FUNCTION_BLOCK "GCS7_E_DEVC"	// FB 38
TITLE = DevCtrl
//  
//COPYRIGHT:    (C) 2004 BY  BUHLER AG, CH-9240 UZWIL  SWITZERLAND
//
//PRODUCT:      GCS7
//
//TITLE:        Element DevCTRL (Profibus)
//              (GCPROVB Revision 10)
//
//-------------------------------------------------------------------------
//
//IDENT:        AUTHOR:             DEPT:                      DATE:
//FB38.2.1      A.Egli              CT3                        01-Dec-2005
//              Parameter Upload Change DBD86-->DBD88
//FB38.2.0      A.Egli              CT3                        05-Jan-2005
//              Parameter Upload (uses DB10)
//FB38.1.1      A. Egli             CT3                        20-Sep-2004
//              Integration test
//FB38.1.0      A. Egli             CT3                        08-Jun-2004
//              1st Release in S7
//
//-------------------------------------------------------------------------
//
//PURPOSE:      MANUAL : see [DEVCENMAN]
//
//RESTRICTIONS: S7
//
//              (*2) : Not used for MZDE
//
//=======================================================
//Log Message: 
//------------------------------------------------------
//0     = Fault Cannceled
//1..79 = AlarmLC : Alarmnumber see manual of MEAF
//90    = Fault Remote Control
//91    = StStopped
//92    = StDosing
//93    = StEmptied
//94    = Timeout starting
//95    = Wrong value
//96    = Communication fault
//97    = 
//98    = 
//99    = Collected alarm
//
//=======================================================
//StCode:  State               
//------------------------------------------------------
//32    StFault                 
// 1    StStopped                   Stopped
//41    Stopped.HWStop              StStopped + InHWStop 
//51    Stopped.DPFault             StStopped + DPFault
// 2    StStarting              
// 3    StStarted               
// 7    StStopping              
//
//
AUTHOR : EA
FAMILY : GCS7LL
NAME : DEVCTRL
VERSION : 2.1
VAR
  StCode : INT ;	//Element state code
  InEnable : BOOL ;	//Enable to run the element (manual and automatic mode)
  InAutomaticControl : BOOL ;	//1=Automatic Control, 0=Manual Control
  CmdRestart : BOOL ;	//Pulse to send "Newstart" to LC
  InHoldStartValue : BOOL ;	//Is sent to LC : de: Startwert aktiv
  spare0203 : BOOL ;
  spare0205 : BOOL ;
  spare0206 : BOOL ;
  spare0207 : BOOL ;
  CmdOff : BOOL ;	//Pulse to stop the element (manual mode)
  CmdOn : BOOL ;	//Pulse to start the element (manual mode)
  CmdNext : BOOL ;	//Pulse to start the element in automatic mode
  CmdFaultReset : BOOL ;	//Command to reset fault
  InLocal : BOOL ;	//1= Local mode (no fault by start with service switch)
  InManual : BOOL ;	//1= Manual / 0= Automatic
  InReport : BOOL ;	//Report of all state transitions
  spare0307 : BOOL ;
  InHWStop : BOOL ;	//HW stop is detected, no fault
  InDPFault : BOOL ;	//DP-Fault is detected, no fault
  InSimulation : BOOL ;	//MZAH: Simulation with DPSim
  OutComFault : BOOL ;	//Communication fault
  OutWrongValue : BOOL ;	//Wrong nominal values, rejected by MEAF
  OutSteamValueOn : BOOL ;	//de: Dampfventil angesteuert
  OutLS1Closed : BOOL ;	//de: Endschalter 1 geschlossen
  OutLS2Closed : BOOL ;	//de: Endschalter 2 geschlossen
  StStopped : BOOL ;	//Element is stopped
  StStarting : BOOL ;	//Element is starting
  StStarted : BOOL ;	//Element is dosing
  StStopping : BOOL ;	//Element is stopping
  StFault : BOOL ;	//Element has a communication or device fault
  InTemperature : INT ;	//Is sent to LC: Target value [0.1°C]  sent to MEAF
  InSteamValueManual : INT ;	//Is sent to LC: Target value steam control manual mode [0.1%]
  InProductFlowrate : DINT ;	//Is sent to LC: Actual flowrate product [kg/h]
  InStartValueSteam : INT ;	//Is sent to LC: CTRL.START Start value for steam control [0.1%]
  InQMin : INT ;	//Is sent to LC: Minimum dosing value TCON.QMIN
  InQMax : INT ;	//Is sent to LC: Maximum dosing value TCON.QMAX
  spare20 : INT ;
  spare22 : INT ;
  spare24 : INT ;
  spare26 : INT ;
  OutTemperature1 : INT ;	//Is read from LC: [0.1°C]
  OutTemperature2 : INT ;	//Is read from LC: [0.1°C]
  OutTemperature3 : INT ;	//Is read from LC: [0.1°C]
  OutSteamAc : DINT ;	//Is read from LC: Actual flowrate steam [0.1%]
  OutStartValueSteam : DINT ;	//Is read from LC: Start value for steam control [0.1%]
  spare42 : DINT ;	//Is read from LC: Minimum dosing value TCON.QMIN
  spare46 : DINT ;	//Is read from LC: Maximum dosing value TCON.QMAX
  OutAlarmNr : INT ;	//Is read from MEAF
  OutAlarmNrLog : INT ;	//Last textnumber send to log
  InFilter : ARRAY  [0 .. 95 ] OF //These alarms are not printed  (1=no alarm)
  BOOL ;
  Par : STRUCT
   ParObjectNo : INT ;	//Is used for communication with PC, e.g. for message
   ParMsgType : INT ;	//Is used for message (translation of state)
   ParHornCode : INT ;	//Is used by horn module
   ParLogOff : BOOL ;	//Report is off
   ParManual : BOOL ;	//Manual mode wihout interlocking
   ParIOByteNr : INT ;	//PROFIBUS: Address of first input and output byte
   ParMonTime : INT ;	//Monitoring time starting and stopping
   OutMonTime : INT ;	//Monitoring time starting and stopping
   OutHelpFlags : STRUCT 	//Is sent to FBAL
    OutAlarmTimeOut : BOOL ;
    CmdFaultReset : BOOL ;
    OutFaultResetDone : BOOL ;
    OutTestNewAlarm : BOOL ;	//Aux. signal to retry fault message
    OutFlagFaultResetDone : BOOL ;
    OutComFaultRead : BOOL ;
    OutComFaultSend : BOOL ;
    OutRelevantFault : BOOL ;
    OutNoAlarm : BOOL ;	//Alarmnumber 0 is read form LC
   END_STRUCT ;
   Command : STRUCT
    Start : BOOL ;	//de: Start
    Automatic : BOOL ;	//de: Automat/Manual
    Restart : BOOL ;	//de: Neustart mit Startwert und Startzeit
    StartValueActive : BOOL ;	//de: Startwert aktiv
    spare04 : BOOL ;
    spare05 : BOOL ;
    spare06 : BOOL ;
    AcceptNewDataReady : BOOL ;	//FBAL: de: Quittierung neue Werte Bereit
    spare10 : BYTE ;
    spare20 : BYTE ;
    CommandReady : BOOL ;	//de: Steuersignale gültig
    spare31 : BOOL ;
    spare32 : BOOL ;
    spare33 : BOOL ;
    spare34 : BOOL ;
    ResetAlarm : BOOL ;	//de: Alarm löschen
    NewSendData : BOOL ;	//de: Aenderung Sendedaten
    AcceptNewRcvData : BOOL ;	//de: Quittierung Aenderung Empfangsdatensatz
   END_STRUCT ;
   Status : STRUCT
    Operation : BOOL ;	//de: Betrieb
    spare01 : BOOL ;
    RestartDone : BOOL ;	//de: Neustart wurde vorgenommen
    spare03 : BOOL ;
    spare04 : BOOL ;
    spare05 : BOOL ;	//
    spare06 : BOOL ;
    NewDataReady : BOOL ;	//de: Neue Werte Bereit
    SteamValueOn : BOOL ;	//de: Dampfventil angesteuert
    LS1Closed : BOOL ;	//de: Endschalter 1 geschlossen
    LS2Closed : BOOL ;	//de: Endschalter 2 geschlossen
    spare20 : BYTE ;
    spare30 : BOOL ;
    spare31 : BOOL ;
    spare32 : BOOL ;
    RemoteControl : BOOL ;	//de: Sollwertvorgabe Remote
    WrongValue : BOOL ;	//de: Falscher Sollwert
    SumFault : BOOL ;	//de: Sammelalarm
    AcceptNewSendData : BOOL ;	//de: Quittierung Aenderung Sendedaten
    NewRcvData : BOOL ;	//de: Aenderung Empfangsdaten
   END_STRUCT ;
  END_STRUCT ;
END_VAR
VAR_TEMP
  tmpLOGvalue : WORD ;	//LOG value
  tmpCommand : INT ;
  tmpFault : BOOL ;
  tmpOff : BOOL ;
  tmpOn : BOOL ;
  tmpLocal : BOOL ;
  tmpLocalFault : BOOL ;
  tmpReport : BOOL ;
  tmpFlag : BOOL ;
  tmpLenDyn : DINT ;
  tmpAddrOffset : DINT ;
  tmpAddr : WORD ;
  tmpReturn : INT ;
  DPData : STRUCT
   StatusCommand : DWORD ;
   NrSndDataSet : BYTE ;	//de: Nummer Sendedatensatz
   IdxSndDataSet : BYTE ;	//de: Index Sendedatensatz
   NrRcvDataSet : BYTE ;	//de: Nummer Empfangsdatensatz
   IdxRcvDataSet : BYTE ;	//de: Index Empfangsdatensatz
   Data : ARRAY  [1 .. 4 ] OF DINT ;
  END_STRUCT ;
  Set001 : STRUCT
   Temperature1 : INT ;	//Is read from LC: [0.1°C]
   Temperature2 : INT ;	//Is read from LC: [0.1°C]
   Temperature3 : INT ;	//Is read from LC: [0.1°C]
   StreamAc : DINT ;	//Is read from LC: Actual flowrate steam [0.1%]
   StartValueSteam : INT ;	//Is read from LC: Start value for steam control [0.1%]
   DosingValueMax : INT ;	//Is read from LC: Maximum dosing value TCON.QMAX
   DosingValueMin : BYTE ;	//Is read from LC: Minimum dosing value TCON.QMIN
   AlarmNr : BYTE ;	//Is read from MEAF
  END_STRUCT ;
  Set128 : STRUCT
   Temperature : INT ;	//Is sent to LC: Target value [0.1°C]  sent to MEAF
   SteamValueManual : INT ;	//Is sent to LC: Target value steam control manual mode [0.1%]
   spare12 : INT ;	//Is sent to LC: Target value steam control manual mode [0.1%]
   FlowrateProdAc : DINT ;	//Is sent to LC: Actual flowrate product [kg/h]
   StartValueSteam : INT ;	//Is sent to LC: CTRL.START Start value for steam control [0.1%]
   DosingValueMax : INT ;	//Is sent to LC: Maximum dosing value TCON.QMAX
   DosingValueMin : INT ;	//Is sent to LC: Minimum dosing value TCON.QMIN
  END_STRUCT ;
END_VAR
BEGIN
NETWORK
TITLE =  Start Global
      L     90;
      T     #tmpLenDyn;	//--> Len dynamic data in byte
      TAR2;
      L     DW#16#FFFFFF;
      AD;
      T     #tmpAddrOffset;
NETWORK
TITLE = PC Control
//=== Test Object number =====================
      L     "SYS_DirectCtrlDB".PC.ObjectNo;	//PCControl.ObjectNo
      L     #Par.ParObjectNo;	//Input ObjectNo
      <>I;
      JC    Ctrl;
//=== Test OType      ========================
      L     1138;	//Input object type
      L     "SYS_DirectCtrlDB".PC.ObjectType;	//PCControl.ObjectType
      <>I;
      JC    Ctrl;
//=== Test Handshake =========================
      A     "SYS_DirectCtrlDB".PC.Hsk.FExamine;	//Handshake.FExamine
      JC    pExa;
      A     "SYS_DirectCtrlDB".PC.Hsk.FDefineCmd;	//Handshake.FDefineCmd
      JC    pCmd;
      A     "SYS_DirectCtrlDB".PC.Hsk.FDefinePara;	//Handshake.FDefinePara
      JC    pPar;
pIni: L     2;	//FcInit
      UC    "SYS_DirectCtrl";
      JU    Ctrl;
//Write parameter 
pPar: NOP   0;
//Write new commands from PC to Interface of group 
pCmd: A     "SYS_DirectCtrlDB".PC.Cmd1[2];	//Cmd1[2]  =CmdRestart
      S     #CmdRestart;
      A     "SYS_DirectCtrlDB".PC.Cmd1[8];	//Cmd1[8]  =CmdOff
      S     #CmdOff;
      A     "SYS_DirectCtrlDB".PC.Cmd1[9];	//Cmd1[9]  =CmdOn
      S     #CmdOn;
      A     "SYS_DirectCtrlDB".PC.Cmd1[10];	//Cmd1[10] =CmdNext
      S     #CmdNext;
      A     "SYS_DirectCtrlDB".PC.Cmd1[11];	//Cmd1[11] =CmdFaultReset
      S     #CmdFaultReset;
      A     "SYS_DirectCtrlDB".PC.Cmd1[13];	//Cmd1[13] =CmdManualOn
      S     #InManual;
      A     "SYS_DirectCtrlDB".PC.Cmd2[13];	//Cmd2[13] =CmdManualOff
      R     #InManual;
      A     "SYS_DirectCtrlDB".PC.Cmd1[14];	//Cmd1[14] =CmdReportOn
      S     #InReport;
      A     "SYS_DirectCtrlDB".PC.Cmd2[14];	//Cmd2[14] =CmdReportOff
      R     #InReport;
//Define Value
      AN    "SYS_DirectCtrlDB".PC.Hsk.FDefineValue;	// PC.Hsk.FDefineValue
      ON    #InManual;
      JC    pIni;
      JU    pIni;
pExa: TAR2;	//Address dynamic datas
      T     "SYS_DirectCtrlDB".GC.InDynAddr;	//-->PCControl.GC.InDynAddr
      L     #tmpLenDyn;	//Length dynamic datas
      T     "SYS_DirectCtrlDB".GC.InDynLen;	//-->PCControl.GC.InDynLen
      L     0;
      T     "SYS_DirectCtrlDB".GC.InParaAddr;	//-->PCControl.GC.InParaAddr
      T     "SYS_DirectCtrlDB".GC.InParaLen;	//-->PCControl.GC.InParaLen
      L     1;	//Code FcExamine
      UC    "SYS_DirectCtrl";
      L     10;	//Revision
      T     "SYS_DirectCtrlDB".GC.Revision;
Ctrl: NOP   0;
NETWORK
TITLE = (Profibus) Read data and store Data 
      L     #Par.ParIOByteNr;
      T     #tmpAddr;
      A     #InSimulation;
      JC    rSim;
      CALL  "SIEMENS_DPRD_DAT" (
           LADDR                    := #tmpAddr,
           RET_VAL                  := #tmpReturn,
           RECORD                   := #DPData);
      L     #tmpReturn;
      L     0;
      <>I;
      =     #Par.OutHelpFlags.OutComFaultRead;
      JC    rcv0;
      JU    rDP;
//read from Simulation
rSim: R     #Par.OutHelpFlags.OutComFaultRead;
      A     "GCS7_Gr_SimDPtoImage";
      L     P#I 0.0;
      JC    rDB1;
      OPN   "TEST_IOSimuliInput";
      L     P#DBX 0.0;
rDB1: L     #Par.ParIOByteNr;
      SLD   3;
      +D;
      LAR1;
      L     D [AR1,P#0.0];
      T     #DPData.StatusCommand;
      L     B [AR1,P#4.0];
      T     #DPData.NrSndDataSet;
      L     B [AR1,P#5.0];
      T     #DPData.IdxSndDataSet;
      L     B [AR1,P#6.0];
      T     #DPData.NrRcvDataSet;
      L     B [AR1,P#7.0];
      T     #DPData.IdxRcvDataSet;
      L     D [AR1,P#8.0];
      T     #DPData.Data[1];
      L     D [AR1,P#12.0];
      T     #DPData.Data[2];
      L     D [AR1,P#16.0];
      T     #DPData.Data[3];
      L     D [AR1,P#20.0];
      T     #DPData.Data[4];
//==Copy Status===============
rDP:  L     #DPData.NrRcvDataSet;
      L     0;
      ==I;
      JC    R001;
      CALL  "SIEMENS_BLKMOV" (
           SRCBLK                   := #DPData.StatusCommand,
           RET_VAL                  := #tmpReturn,
           DSTBLK                   := #Par.Status);
      AN    #Par.Status.NewRcvData;
      A     #InSimulation;
      JC    rcv0;
//===============================
//Answer Dataset 001
      L     #DPData.NrRcvDataSet;
      L     1;
      <>I;
      JC    r11;	//[2.0]
      CALL  "SIEMENS_BLKMOV" (
           SRCBLK                   := #DPData.Data,
           RET_VAL                  := #tmpReturn,
           DSTBLK                   := #Set001);
      L     #Set001.Temperature1;
      T     #OutTemperature1;
      L     #Set001.Temperature2;
      T     #OutTemperature2;
      L     #Set001.Temperature3;
      T     #OutTemperature3;
      L     #Set001.StreamAc;
      T     #OutSteamAc;
      L     #Set001.StartValueSteam;
      T     #OutStartValueSteam;
//Reset old alarm flags with CmdFaultReset
      A     #Par.OutHelpFlags.OutFlagFaultResetDone;
      A     "SYS_Pulse1000ms";
      R     #Par.OutHelpFlags.OutFlagFaultResetDone;
      R     #Par.OutHelpFlags.OutFaultResetDone;
      S     #Par.OutHelpFlags.OutTestNewAlarm;
      L     0;
      L     #Set001.AlarmNr;
      ==I;
      =     #Par.OutHelpFlags.OutNoAlarm;
//  keep old alalrm number
      A     #Par.OutHelpFlags.OutNoAlarm;
      A     #Par.OutHelpFlags.OutRelevantFault;
      AN    #Par.OutHelpFlags.OutTestNewAlarm;
      AN    #InLocal;
      AN    #InManual;
      JC    rA1;
      T     #OutAlarmNr;
rA1:  JU    R11;	//[2.0]   
//===============================
//[2.0]--> LC Parameter 
//Reading dataset 11
R11:  L     "SYS_DirectCtrlLCDB".PC.ObjectNo;
      L     #Par.ParObjectNo;
      <>I;
      JC    R127;
      AN    "SYS_DirectCtrlLCDB".PC.Hsk.FExamineFirst;
      AN    "SYS_DirectCtrlLCDB".PC.Hsk.FExamineNext;
      JC    R127;
// -- Start Reading with Dataset 11
      L     11;
      T     #DPData.NrRcvDataSet;
      L     253;	//First
      A     "SYS_DirectCtrlLCDB".PC.Hsk.FExamineFirst;
      JC    rLC9;
      L     254;	//Next
rLC9: T     #DPData.IdxRcvDataSet;
      JU    rcv0;
//---Answer  dataset 11 ---
//---Answer  dataset 12 ---
r11:  L     #DPData.NrRcvDataSet;
      L     11;
      <>I;
      JC    rLCB;
// Answer Dataset 11
      L     '  ';
      T     "SYS_DirectCtrlLCDB".PC.Value[1];
      L     #DPData.Data[1];
      T     DB10.DBD 60;
      L     #DPData.Data[2];
      T     DB10.DBD 64;
      L     #DPData.Data[3];
      T     DB10.DBD 68;
      L     #DPData.Data[4];
      T     DB10.DBD 72;
      L     #DPData.IdxRcvDataSet;
      L     255;
      ==I;
      JC    rLCE;
      S     "SYS_DirectCtrlLCDB".GC.Set11Done;
      L     12;
      T     #DPData.NrRcvDataSet;
      L     0;
      T     #DPData.IdxRcvDataSet;
      JU    rcv0;	//--> Read dataset 12
// Answer Dataset 12
rLCB: L     #DPData.NrRcvDataSet;
      L     12;
      <>I;
      JC    r127;
      L     #DPData.Data[1];
      T     DB10.DBD 76;
      L     #DPData.Data[2];
      T     DB10.DBD 80;
      L     #DPData.Data[3];
      T     DB10.DBD 84;
      L     #DPData.Data[4];
      T     DB10.DBD 88;
      AN    "SYS_DirectCtrlLCDB".GC.Set11Done;
      JC    R127;
rLCE: L     12;
      CALL  "SYS_DirectCtrl";
      JU    R127;
//<--[2.0]
//===============================
//Answer  dataset 127
r127: L     #DPData.NrRcvDataSet;
      L     127;
      <>I;
      JC    r001;
      JU    R001;
//===============================
//Else Read Dataset 1
r001: JU    R001;	// =no valide answer read dataset 001
//===============================
//Read Dataset 001
R001: L     1;
      T     #DPData.NrRcvDataSet;
      L     0;
      T     #DPData.IdxRcvDataSet;
      A     #Par.OutHelpFlags.OutFaultResetDone;
      AN    "SYS_Pulse1000ms";
      S     #Par.OutHelpFlags.OutFlagFaultResetDone;
      JU    rcv0;
//===============================
//Read Dataset 127
R127: L     127;
      T     #DPData.NrRcvDataSet;
      L     0;
      T     #DPData.IdxRcvDataSet;
      JU    rcv0;
//===============================
rcv0: NOP   0;
NETWORK
TITLE = (Profibus) Status to ASW
      A     #Par.OutHelpFlags.OutComFaultRead;
      O     #Par.OutHelpFlags.OutComFaultSend;
      =     #OutComFault;
      A     #Par.Status.SteamValueOn;
      AN    #OutComFault;
      =     #OutSteamValueOn;
      A     #Par.Status.LS1Closed;
      AN    #OutComFault;
      =     #OutLS1Closed;
      A     #Par.Status.LS2Closed;
      AN    #OutComFault;
      =     #OutLS2Closed;
//=======================================
//Init in local mode  
//=======================================
      AN    #InLocal;
      AN    #InManual;
      ON    #OutComFault;
      JC    alJL;
      L     0;
      T     #OutSteamAc;
alJL: NOP   0;
NETWORK
TITLE =  All State Init
//===Clear tmp Variable
//===Global Group Orders===
      A     "GCS7_Gr_OutManualOn";	//Global.OutManualOn
      S     #InManual;
      A     "GCS7_Gr_OutManualOff";	//Global.OutManualOff
      R     #InManual;
      A     #InManual;
      S     "GCS7_Gr_InManual";	//Global.InManualMode
//---Report is on---
      O     "GCS7_Gr_OutReportAll";	//---Global OutReportAll
      O     #InReport;
      =     #tmpReport;
//---FaultReset is on---
      A     "GCS7_Gr_OutFaultReset";	//Gr.OutFaultReset
      S     #CmdFaultReset;
//---State---
//---Local---
      A     #InLocal;
      AN    #InManual;
      =     #tmpLocalFault;
      A     #tmpLocalFault;
      O     #InHWStop;
      O     #InDPFault;
      =     #tmpLocal;
//---Off---
      AN    #InManual;
      ON    #Par.ParManual;
      AN    #InEnable;
      O     #tmpLocal;
      O     #CmdOff;
      =     #tmpOff;
//---On---
      A     #CmdNext;
      AN    #InManual;
      O     #CmdOn;
      AN    #tmpOff;
      =     #tmpOn;
//--- Time out---
      AN    #StStarting;
      AN    #StStopping;
      AN    #StFault;
      R     #Par.OutHelpFlags.OutAlarmTimeOut;
      JC    inJ1;
      A     #Par.OutHelpFlags.OutAlarmTimeOut;
      O     #StFault;
      JC    inJ1;
      L     0;
      L     #Par.OutMonTime;
      >I;
      =     #Par.OutHelpFlags.OutAlarmTimeOut;
      AN    "GCS7_Gr_OutTick200ms";	// Global Tick 200ms
      JC    inJ1;
      +     -2;	// Decrement all 200ms
      T     #Par.OutMonTime;
inJ1: NOP   0;
//=======================================
//Fault   
//=======================================
      A     #Par.Status.WrongValue;
      =     #OutWrongValue;
//--- Fault   
      LAR1  #tmpAddrOffset;
      L     P##InFilter;
      +AR1;	//Pointer to #InFilter
      L     #OutAlarmNr;
      +AR1;	//Pointer to #InFilter[OutAlarmNumber]
      L     #OutAlarmNr;
      L     0;
      <>I;
      AN    DIX [AR1,P#0.0];	//#InFilter[OutAlarmNumber]
      O;
      A     #Par.Status.SumFault;
      AN    #InFilter[0];
      =     #Par.OutHelpFlags.OutRelevantFault;
      A     #Par.OutHelpFlags.OutRelevantFault;
      A     #Par.Status.SumFault;
      O     #OutComFault;
      O     #Par.OutHelpFlags.OutAlarmTimeOut;
      O     #Par.Status.WrongValue;
      ON    #Par.Status.RemoteControl;
      AN    #tmpLocal;
      =     #tmpFault;
NETWORK
TITLE = (Profibus) Prepare Command for MEAF
      A     #Par.Command.Start;
      =     #tmpFlag;
      A     #tmpOn;
      S     #Par.Command.Start;
      A     #StFault;
      O     #tmpOff;
      O     #StStopping;
      R     #Par.Command.Start;
//==============================
      A     #InAutomaticControl;
      =     #Par.Command.Automatic;
//================================
      A     #CmdRestart;
      S     #Par.Command.Restart;
      A     #CmdRestart;
      A     #Par.Command.Restart;
      A     #Par.Status.RestartDone;
      R     #Par.Command.Restart;
      R     #CmdRestart;
//================================
      A     #InHoldStartValue;
      =     #Par.Command.StartValueActive;
//==============================
      A     #Par.Status.AcceptNewSendData;
      A     #Par.Command.ResetAlarm;
      R     #Par.Command.ResetAlarm;
      S     #Par.OutHelpFlags.OutFaultResetDone;
      A     #CmdFaultReset;
      AN    #Par.Status.AcceptNewSendData;
      R     #CmdFaultReset;
      S     #Par.Command.ResetAlarm;
      R     #Par.OutHelpFlags.OutAlarmTimeOut;
//==============================
      A     #Par.Status.NewDataReady;
      =     #Par.Command.AcceptNewDataReady;
//==============================
      SET;
      =     #Par.Command.CommandReady;
//==============================
      A     #Par.Status.NewRcvData;
      =     #Par.Command.AcceptNewRcvData;
//==============================
      AN    #Par.Status.AcceptNewSendData;
      =     #Par.Command.NewSendData;
NETWORK
TITLE = (Profibus) Send Data
//======================================================
//Test Send Dataset 000 done
      L     #DPData.NrSndDataSet;
      L     0;
      <>I;
      JC    s128;
      JU    S128;	//-->send 128
//------------------------------------------------
//Test Send Dataset 128 done
s128: L     #DPData.NrSndDataSet;
      L     128;
      <>I;
      JC    S000;	//-->Send 000
      JU    S128;	//-->Send 128
//==================================================
//Send Dataset 128
S128: L     128;
      T     #DPData.NrSndDataSet;
      L     0;
      T     #DPData.IdxSndDataSet;
      L     #InTemperature;
      T     #Set128.Temperature;
      L     #InSteamValueManual;
      T     #Set128.SteamValueManual;
      L     0;
      T     #Set128.spare12;
      L     #InProductFlowrate;
      T     #Set128.FlowrateProdAc;
      L     #InStartValueSteam;
      T     #Set128.StartValueSteam;
      L     #InQMax;
      T     #Set128.DosingValueMax;
      L     #InQMin;
      T     #Set128.DosingValueMin;
      JU    send;
//======================================================
//Send Dataset 0
S000: L     0;
      T     #DPData.NrSndDataSet;
      L     0;
      T     #DPData.IdxSndDataSet;
send: CALL  "SIEMENS_BLKMOV" (
           SRCBLK                   := #Par.Command,
           RET_VAL                  := #tmpReturn,
           DSTBLK                   := #DPData.StatusCommand);
      CALL  "SIEMENS_BLKMOV" (
           SRCBLK                   := #Set128,
           RET_VAL                  := #tmpReturn,
           DSTBLK                   := #DPData.Data);
      A     #InSimulation;
      JC    sSim;
      CALL  "SIEMENS_DPWR_DAT" (
           LADDR                    := #tmpAddr,
           RECORD                   := #DPData,
           RET_VAL                  := #tmpReturn);
      L     #tmpReturn;
      L     0;
      <>I;
      =     #Par.OutHelpFlags.OutComFaultSend;
      JU    DP_C;
//write to Simulation
sSim: R     #Par.OutHelpFlags.OutComFaultSend;
      A     "GCS7_Gr_SimDPtoImage";
      L     P#Q 0.0;
      JC    rDB2;
      OPN   "TEST_IOSimuliOutput";
      L     P#DBX 0.0;
rDB2: L     #Par.ParIOByteNr;
      SLD   3;
      +D;
      LAR1;
      L     #DPData.StatusCommand;
      T     D [AR1,P#0.0];
      L     #DPData.NrSndDataSet;
      T     B [AR1,P#4.0];
      L     #DPData.IdxSndDataSet;
      T     B [AR1,P#5.0];
      L     #DPData.NrRcvDataSet;
      T     B [AR1,P#6.0];
      L     #DPData.IdxRcvDataSet;
      T     B [AR1,P#7.0];
      L     #DPData.Data[1];
      T     D [AR1,P#8.0];
      L     #DPData.Data[2];
      T     D [AR1,P#12.0];
      L     #DPData.Data[3];
      T     D [AR1,P#16.0];
      L     #DPData.Data[4];
      T     D [AR1,P#20.0];
DP_C: NOP   0;
NETWORK
TITLE = States
//===State machine===
      A     #StStopped;
      JC    S0;
      A     #StStarting;
      JC    S1;
      A     #StStarted;
      JC    S2;
      A     #StStopping;
      JC    S3;
      A     #StFault;
      JC    S4;
      S     #StStopped;	//Init
      JU    S0;
NETWORK
TITLE =  StStopped
xxS0: S     #StStopped;
      R     #StStarted;
      JU    LOGX;
S0:   A     #tmpFault;
      R     #StStopped;
      JC    xxS4;	//--> Transition to StFault
      A     #Par.Status.Operation;
      AN    #OutComFault;
      O     #Par.Command.Start;
      R     #StStopped;
      JC    xxS1;	//--> Transition to StStarting
      JU    OUT;
NETWORK
TITLE =  StStarting
xxS1: S     #StStarting;
      R     #Par.OutHelpFlags.OutAlarmTimeOut;
      L     #Par.ParMonTime;
      T     #Par.OutMonTime;
      JU    OUT;
S1:   A     #tmpFault;	//Condition for StFault
      R     #StStarting;
      JC    xxS4;	//--> Transition to StFault
      A     #tmpOff;
      R     #StStarting;
      JC    xxS3;	//--> Transition to StStopping
      A     #Par.Status.Operation;
      R     #StStarting;
      JC    xxS2;	//--> Transition to StStarted
      JU    OUT;
NETWORK
TITLE =  StStarted
xxS2: S     #StStarted;
      JU    LOGX;
S2:   A     #tmpFault;	//Condition for StFault/StFalse
      R     #StStarted;
      JC    xxS4;	//--> Transition to StFault
      A     #tmpOff;
      ON    #Par.Status.Operation;
      R     #StStarted;
      JC    xxS3;	//--> Transition to StStopping
      JU    OUT;
NETWORK
TITLE =  StStopping
xxS3: S     #StStopping;
      R     #Par.OutHelpFlags.OutAlarmTimeOut;
      L     #Par.ParMonTime;
      T     #Par.OutMonTime;
      A     #StFault;
      R     #StFault;
      JC    LOGC;	//-->Message Operator ('fault cancelled' )
//State StStopping
S3:   A     #tmpFault;
      AN    #tmpLocal;
      R     #StStopping;
      JC    xxS4;	//-->Transition to StFault
      A     #tmpOn;
      R     #StStopping;
      JC    xxS1;	//-->Transition to StStarting 
      AN    #Par.Status.Operation;
      O     #OutComFault;
      R     #StStopping;
      JC    xxS0;	//-->Transition to StStopped 
      JU    OUT;
NETWORK
TITLE =  FAULT
// State Fault
S4:   AN    #tmpFault;	//---Condition for StStopping
      A     #Par.OutHelpFlags.OutTestNewAlarm;
      O     #tmpLocalFault;
      JC    xxS3;	// Transition to StStopping
      A     #Par.OutHelpFlags.OutTestNewAlarm;
      JC    xxS4;
      JU    OUT;
NETWORK
TITLE = LOG
xxS4: S     "GCS7_Gr_InFaultFlag";	//Gr.InFaultFlag
      S     #StFault;
      R     #Par.OutHelpFlags.OutFaultResetDone;
      R     #Par.OutHelpFlags.OutTestNewAlarm;
      CALL  "SYS_Horn_Code" (
           FcCode                   := 1,
           ParObjectType            := 1138,
           ParObjectNo              := #Par.ParObjectNo,
           ParHornCode              := #Par.ParHornCode);
      L     #Par.ParMonTime;
      T     #Par.OutMonTime;
//Alarm Communication
      L     B#(1, 96);
      A     #OutComFault;
      JC    LOG;
//Tiemout
      A     #Par.OutHelpFlags.OutAlarmTimeOut;
      L     B#(1, 94);	// Message ('fault timeout')
      JC    LOG;
//Alarm-Nr 1..80
      L     0;
      L     #OutAlarmNr;
      ==I;
      JC    LOG2;
      L     B#(1, 0);
      OW;
      JU    LOG;	//Alarms 1..80
//Fault Remote Control
LOG2: L     B#(1, 90);	// Message ('fault DP Mode')   //[5.2]
      AN    #Par.Status.RemoteControl;	//[5.2]
      JC    LOG;	//[5.2]
//Fault Wrong Value
      A     #Par.Status.WrongValue;
      L     B#(1, 95);	// Message ('fault wrong value')
      JC    LOG;
//Collected Alarm
      L     B#(1, 99);	// Message ('fault collected alarm')
      JU    LOG;
//===============================================
//State Transition
LOGX: AN    #tmpReport;
      JC    OUT;
      A     #StStopped;
      L     B#(4, 91);	//Message ('Stopped')
      JC    LOG;
      A     #StStarted;
      L     B#(4, 92);	//Message ('Started')
      JC    LOG;
      JU    OUT;
LOGC: L     B#(4, 0);	//Message ('fault cancelled')
LOG:  A     #Par.ParLogOff;	//---Set LOG Message
      JC    OUT;
      T     #tmpLOGvalue;
      L     W#16#FF;
      AW;
      T     #OutAlarmNrLog;
      CALL  "GCS7_LogConvert" (
           ObjectNo                 := #Par.ParObjectNo,
           MsgType                  := #Par.ParMsgType,
           ClassMsgTxt              := #tmpLOGvalue,
           OType                    := 1138);	//LOG Message Converter / Entry / Contains Class and TextNo
NETWORK
TITLE = Global End
OUT:  SET;	//---Clear all commands
      R     #CmdOff;
      R     #CmdOn;
      R     #CmdNext;
//--Output for group 
      AN    #InLocal;
      O     #InManual;
      A     #InDPFault;
      S     "GCS7_Gr_InDPFault";
      AN    #InLocal;
      O     #InManual;
      A     #InHWStop;
      S     "GCS7_Gr_InHWStop";
NETWORK
TITLE = State Code
//--Stopped, Substate ---
      AN    #StStopped;
      JC    STC2;
      L     41;	//Code: StStopped.HWStop
      A     #InHWStop;
      JC    STC;
      L     51;	//Code: StStopped.DPFault
      A     #InDPFault;
      JC    STC;
      L     1;	// Code: stopped
      JC    STC;
//--------------------
STC2: L     2;	//Code: StStarting
      A     #StStarting;
      JC    STC;
      L     3;	//Code: StStarted
      A     #StStarted;
      JC    STC;
      L     7;	//Code: StStopping
      A     #StStopping;
      JC    STC;
      L     32;	//Code: fault
STC:  L     #StCode;	//Old state code
      TAK;
      T     #StCode;	//Save state code
      <>I;
      L     3;	//Load code for CBit methode
      CC    "SYS_CBitCtrl";
END_FUNCTION_BLOCK

FUNCTION_BLOCK "GCS7_E_MYFA_MOZD"	// FB 39
TITLE = MYFA-MOZD
//  
//COPYRIGHT:    (C) 1997  BUHLER AG, CH-9240 UZWIL, SWITZERLAND
//
//PRODUCT:      GCS7
//
//TITLE:        Element Control MYFA-MOZD or MOZD (Liquid Regulator)
//
//-------------------------------------------------------------------------
//
//IDENT:        AUTHOR:             DEPT:                       DATE:
//
//FB39.3.0      A. Egli             CT3                         17-Jun-2002
//              New Release with one block
//              MOZD or MYFA-MOZD  
//FB39.2.1      A. Egli             CT3                         11-Oct-1999
//              M12.2 "Gr.OutCmdNext removed
//FB39.2A       A. Egli             CT3                         04-Mai-1998
//              StFault = StCode 32
//FB39.1A       A.Egli              AEE61                       25-Jul-1997
//              1st Release in S7
//
//-------------------------------------------------------------------------
//
//PURPOSE:      MANUAL : see [MYFxxMAN]
//
//RESTRICTIONS: S7
//              ACCU2: Pointer to dynamic datas of the element
//              ACCU1: Pointer to parameter datas of the element
//
//-------------------------------------------------------------------------
//=======================================================
//Log Message: 
//------------------------------------------------------
// 0   stopped
// 1   started
// 9   fault cancelled
//10   fault MYFA
//11   fault analog input
//12   fault set value
//
//=======================================================
//StCode:  State               
//------------------------------------------------------
//32   StFault                 
// 1   StStopped               
//41   StStopped.HWStop           StStopped + InHWStop 
//51   StStopped.DPFault          StStopped + DPFault
// 3   StStarted               
//
AUTHOR : EA
FAMILY : GCS7LL
NAME : MYFAMOZD
VERSION : 3.0
VAR
  StCode : INT ;	//Element state code
  InEnable : BOOL ;	//Enable to run
  spare0201 : BOOL ;
  spare0202 : BOOL ;
  spare0203 : BOOL ;
  spare0204 : BOOL ;
  CmdNewJob : BOOL ;	//Pulse to erase OutWtTotalWater
  InRemote : BOOL ;	//Target flowrate for MOZD from PLC
  InpLcOk : BOOL ;	//Digital input 1=MOZD ok / 0=MOZD Alarm
  CmdOff : BOOL ;	//Pulse to start in manual mode
  CmdOn : BOOL ;	//Pulse to stop in manual mode
  CmdNext : BOOL ;	//Start next element (Automatic mode)
  CmdFaultReset : BOOL ;	//Command to reset fault
  InLocal : BOOL ;	//1= Local mode
  InManual : BOOL ;	//1= Manual/ 0= Automatic
  InReport : BOOL ;	//Report of all state transitions
  spare0307 : BOOL ;
  InHWStop : BOOL ;	//HW stop is detected, no fault
  InDPFault : BOOL ;	//DP-Fault is detected, no fault
  OutFaultAI : BOOL ;	//Fault analog input
  OutFaultSetValue : BOOL ;	//Set value out of range
  spare0404 : BOOL ;
  spare0405 : BOOL ;
  OutpRemote : BOOL ;	//Digital output flowrate water from PLC
  spare0407 : BOOL ;
  StStopped : BOOL ;	//Element is stopped
  spare0501 : BOOL ;
  StStarted : BOOL ;	//Element is started
  spare0503 : BOOL ;
  StFault : BOOL ;	//Element has a fault
  InpFlowrateWater : INT ;	//Analog input actual flowrate water [digits]
  MYFA : STRUCT 	//With MYFA
   InMoisture : INT ;	//Moisture target value [0.1 %]
   InpFlowrateProduct : INT ;	//Analog input actual flowrate product [digits]
   InpMoisture : INT ;	//Analog input actual moisture [digits]
   OutMoisture : INT ;	//Moisture actual value [0.1 %]
   OutFlowrateProduct : INT ;	//Flowrate product actual value in [kg/h]
   OutpMoisture : INT ;	//Analog output to target moisture [digits]
  END_STRUCT ;
  MOZD : STRUCT 	//Without MYFA
   InOutFlowrateWaterPpm : INT ;	//Flowrate water target value [0.0 to 10.0%]
   InOutFlowrateWater : INT ;	//Flowrate water target value [dl/h]
   InFlowrateProduct : INT ;	//Flowrate product actual value in [kg/h]
   OutpFlowrateWater : INT ;	//Analog output target flowrate water
   OutpFlowrateProduct : INT ;	//Analog output flowrate product
  END_STRUCT ;
  OutFlowrateWater : INT ;	//Flowrate water actual value in [dl/h]
  OutTotalWater : DINT ;	//Total feeded weight water   [dl]
  OutAlarmNrLog : INT ;	//Last textnumber send to log
  Par : STRUCT
   ParObjectNo : INT ;	//Is used for communication with PC, e.g. for message
   ParMsgType : INT ;	//Is used for message (translation of state)
   ParHornCode : INT ;	//Is used by horn module
   ParLogOff : BOOL ;	//Report is off
   ParManual : BOOL ;	//Manual mode without interlocking
   ParWago : BOOL ;	//Wago analog module format
   ParMYFA : BOOL ;
   ParInFlowrateWaterPc : BOOL ;	//Target value flowrate water from group in Pc
   ParOutFlowrateWaterPc : BOOL ;	//Analog output flowrate water in [0.0 to 10.0%]
   ParFlowrateWater100Pc : INT  := 20000;	//Flowrate water   by 100 % of analog value [dl/h]
   ParFlowrateProduct100Pc : INT  := 30000;	//Flowrate product by 100 % of analog value [kg/h]
   OutCorrectionWeight : REAL ;	//Correction weight for calcuation of OutWtTotalWater [kg]
   spare16 : DINT ;
  END_STRUCT ;
END_VAR
VAR_TEMP
  tmpLOGvalue : WORD ;	//LOG value
  tmpReport : BOOL ;	//Global LOG all
  tmpEnable : BOOL ;
  tmpLenDyn : DINT ;
  tmpEndTime : BOOL ;
  tmpLocal : BOOL ;
  tmpFault : BOOL ;
  tmpFlowWater : REAL ;
  tmpMaxDigits : REAL ;	//ParWago=0: 27'648 / ParWago=1: 32'767
  tmpLocalFault : BOOL ;
END_VAR
BEGIN
NETWORK
TITLE =  Start Global
      L     58;
      T     #tmpLenDyn;	//--> Len dynamic data in byte
NETWORK
TITLE = PC Control
//=== Test Object number =====================
      L     "SYS_DirectCtrlDB".PC.ObjectNo;	//PCControl.ObjectNo
      L     #Par.ParObjectNo;	//Input ObjectNo
      <>I;
      JC    Ctrl;
//=== Test OType      ========================
      L     1039;	//Input object type
      L     "SYS_DirectCtrlDB".PC.ObjectType;	//PCControl.ObjectType
      <>I;
      JC    Ctrl;
//=== Test Handshake =========================
      A     "SYS_DirectCtrlDB".PC.Hsk.FExamine;	// Handshake.FExamine
      JC    pExa;
      A     "SYS_DirectCtrlDB".PC.Hsk.FDefineCmd;	// Handshake.FDefineCmd
      JC    pCmd;
      A     "SYS_DirectCtrlDB".PC.Hsk.FDefinePara;	// Handshake.FDefinePara
      JC    pPar;
pIni: L     2;	// FcInit
      UC    "SYS_DirectCtrl";
      JU    Ctrl;
// Write parameter 
pPar: NOP   0;
// Write new commands from PC to Interface of group 
pCmd: A     "SYS_DirectCtrlDB".PC.Cmd1[8];	//Cmd1[8] =CmdOff
      S     #CmdOff;
      A     "SYS_DirectCtrlDB".PC.Cmd1[9];	//Cmd1[9] =CmdOn
      S     #CmdOn;
      A     "SYS_DirectCtrlDB".PC.Cmd1[10];	//Cmd1[10] =CmdNext
      S     #CmdNext;
      A     "SYS_DirectCtrlDB".PC.Cmd1[11];	//Cmd1[11] =CmdFaultReset
      S     #CmdFaultReset;
      A     "SYS_DirectCtrlDB".PC.Cmd1[13];	//Cmd1[13] =CmdManualOn
      S     #InManual;
      A     "SYS_DirectCtrlDB".PC.Cmd2[13];	//Cmd2[13] =CmdManualOff
      R     #InManual;
      A     "SYS_DirectCtrlDB".PC.Cmd1[14];	//Cmd1[14] =CmdReportOn
      S     #InReport;
      A     "SYS_DirectCtrlDB".PC.Cmd2[14];	//Cmd2[14] =CmdReportOff
      R     #InReport;
      JU    pIni;
pExa: TAR2;	// Address Dynamic datas
      T     "SYS_DirectCtrlDB".GC.InDynAddr;	// -->PCControl.GC.InDynAddr
      L     #tmpLenDyn;	// Length Dynamic datas
      T     "SYS_DirectCtrlDB".GC.InDynLen;	// -->PCControl.GC.InDynLen
      L     0;
      T     "SYS_DirectCtrlDB".GC.InParaAddr;	// -->PCControl.GC.InParaAddr
      T     "SYS_DirectCtrlDB".GC.InParaLen;	// -->PCControl.GC.InParaLen
      L     1;	// Code FcExamine
      UC    "SYS_DirectCtrl";
      L     10;	//Revision
      T     "SYS_DirectCtrlDB".GC.Revision;
NETWORK
TITLE =  All State Init
//===Clear tmp Variable
//===Global Group Orders===
Ctrl: A     "GCS7_Gr_OutManualOn";	//Gr.OutManualOn
      S     #InManual;
      A     "GCS7_Gr_OutManualOff";	//Gr.OutManualOff
      R     #InManual;
      A     #InManual;
      S     "GCS7_Gr_InManual";	//Gr.InManual
//---Local---
      A     #InLocal;
      AN    #InManual;
      =     #tmpLocalFault;
      A     #tmpLocalFault;
      O     #InHWStop;
      O     #InDPFault;
      =     #tmpLocal;
//---Report is on---
      A     "GCS7_Gr_OutReportAll";	//Gr.OutReportAll
      O     #InReport;
      =     #tmpReport;
//---tmpEnable---
      A     #InEnable;
      AN    #InLocal;
      AN    #InManual;
      O(;
      A     #InEnable;
      O     #Par.ParManual;
      A     #InManual;
      );
      AN    #CmdOff;
      =     #tmpEnable;
//---tmpFault---
      L     #MOZD.InOutFlowrateWater;
      L     #Par.ParFlowrateWater100Pc;
      >D;
      O(;
      L     #MOZD.InFlowrateProduct;
      L     #Par.ParFlowrateProduct100Pc;
      >D;
      );
      AN    #Par.ParMYFA;
      O(;
      L     #MYFA.InMoisture;
      L     200;
      >I;
      A     #Par.ParMYFA;
      );
      =     #OutFaultSetValue;
      A     #OutFaultAI;	//Overflow analog input
      ON    #InpLcOk;
      O     #OutFaultSetValue;
      =     #tmpFault;
      A     #InRemote;
      =     #OutpRemote;
//---tmpMaxDigits
      L     2.764800e+04;	//Siemens fullrange MaxDigits
      AN    #Par.ParWago;
      JC    Ctr2;
      L     3.276700e+04;	//Wago fullrange MaxDigits
Ctr2: T     #tmpMaxDigits;
NETWORK
TITLE = States
//===State machine===
      A     #StStopped;
      JC    S0;
      A     #StStarted;
      JC    S2;
      A     #StFault;
      JC    S4;
      S     #StStopped;	// Init
      JU    S0;
NETWORK
TITLE = StStopped
// Any transition to StClosed
xxS0: S     #StStopped;
      AN    #InReport;
      JC    OUT;
      L     B#(4, 0);	// Message ('stopped' )
      JU    LOG;
//=== Logic ====
//Transition to StStarted 
S0:   A     #CmdNext;
      AN    #InManual;
      A     #tmpEnable;
      O;
      A     #CmdOn;
      A     #InManual;
      A     #tmpEnable;
      R     #StStopped;
      JC    xxS2;
//Transition to StFault 
      A     #tmpFault;
      AN    #tmpLocal;
      R     #StStopped;
      JC    xxS4;
      JU    OUT;
NETWORK
TITLE = StStarted
// Any transition to StStarted
xxS2: S     #StStarted;
      S     #StStarted;
      AN    #tmpReport;
      JC    OUT;
      L     B#(4, 1);	// Message ('started')
      JU    LOG;
//=== Logic ====
//Transition to StStopped
S2:   AN    #tmpEnable;
      R     #StStarted;
      JC    xxS0;
// Transition to StFault
      A     #tmpFault;
      AN    #tmpLocal;
      R     #StStarted;
      JC    xxS4;
      JU    OUT;
NETWORK
TITLE = StFault
// Any transiton to Fault  
xxS4: S     "GCS7_Gr_InFaultFlag";	// Gr.InFaultFlag
      S     #StFault;
      CALL  "SYS_Horn_Code" (
           FcCode                   := 1,
           ParObjectType            := 1039,
           ParObjectNo              := #Par.ParObjectNo,
           ParHornCode              := #Par.ParHornCode);
      A     #OutFaultAI;	//Overflow analog input
      L     B#(1, 11);	// Message ('fault analag input' )
      JC    LOG;
      A     #OutFaultSetValue;
      L     B#(1, 12);	//Message ('fault set value' )
      JC    LOG;
      L     B#(1, 10);	// Message ('fault MYFA' )
      JU    LOG;
//=== Logic ====
S4:   AN    #CmdFaultReset;
      AN    "GCS7_Gr_OutFaultReset";	//Gr.OutFaultReset
      AN    #tmpLocal;
      JC    OUT;
// retry of fault message
      A     #tmpFault;
      AN    #tmpLocal;
      JC    xxS4;
      R     #StFault;
      S     #StStopped;
      L     B#(3, 9);	// Message ('fault cancelled' )
      JU    LOG;
NETWORK
TITLE = Log
LOG:  A     #Par.ParLogOff;	//---Set LOG Message
      JC    OUT;
      T     #tmpLOGvalue;
      L     W#16#FF;
      AW;
      T     #OutAlarmNrLog;
      CALL  "GCS7_LogConvert" (
           ObjectNo                 := #Par.ParObjectNo,
           MsgType                  := #Par.ParMsgType,
           ClassMsgTxt              := #tmpLOGvalue,
           OType                    := 1039);	// LOG Message Converter / Entry / Contains Class and TextNo
OUT:  NOP   0;
      SET;
      R     #OutFaultAI;	//--> Overflow analog input
NETWORK
TITLE = MOZD: Calculate target flowrate Water 
      A     #Par.ParInFlowrateWaterPc;
      JC    fwPc;
      L     #MOZD.InOutFlowrateWater;	//[dl/h]
      DTR;
      L     #MOZD.InFlowrateProduct;	//[kg/h]
      DTR;
      /R;
      L     1.000000e+02;	//0.1 *1000                  
      *R;
      RND;
      T     #MOZD.InOutFlowrateWaterPpm;	//-->Target flowrate water in [0.1%] 
      JU    fwJ0;
fwPc: L     #MOZD.InFlowrateProduct;
      DTR;
      L     #MOZD.InOutFlowrateWaterPpm;
      DTR;
      *R;
      L     1.000000e+02;
      /R;
      RND;
      T     #MOZD.InOutFlowrateWater;	//--> Target flowrate water
NETWORK
TITLE = MOZD: Calculate Analog Output value flow water
fwJ0: L     0;
      AN    #StStarted;
      ON    #OutpRemote;
      JC    fwJ1;
      AN    #Par.ParOutFlowrateWaterPc;
      JC    fwJ2;
// Analog output: Unit = 0..10%
      L     #MOZD.InOutFlowrateWaterPpm;	// dl/h
      DTR;	// Integer to real
      L     1.000000e+02;	// 10.0% 
      <=R;
      JC    fwJ3;
      L     1.000000e+00;	// 100%          
      JU    fwJ4;
// Analog output: Unit = dl/h
fwJ2: L     #MOZD.InOutFlowrateWater;	// dl/h
      DTR;	// Integer to real
      L     #Par.ParFlowrateWater100Pc;
      DTR;	// Integer to real
      <=R;
      JC    fwJ3;
      L     1.000000e+00;	// 100%          
      JU    fwJ4;
fwJ3: /R;
fwJ4: L     #tmpMaxDigits;	// Units maximum         
      *R;
      RND;	// Real to Integer
fwJ1: T     #MOZD.OutpFlowrateWater;
NETWORK
TITLE = MOZD:Calculate Analog Output flowrate product
      L     0;
      AN    #StStarted;
      JC    fpJ1;
      L     #MOZD.InFlowrateProduct;	//  kg/h
      DTR;	// Integer to real
      L     #Par.ParFlowrateProduct100Pc;
      DTR;	// Integer to real
      <=R;
      JC    fpJ2;
      L     1.000000e+00;	// 100%          
      JU    fpJ3;
fpJ2: /R;
fpJ3: L     #tmpMaxDigits;	// Units maximum         
      *R;
      RND;	// Real to Integer
fpJ1: T     #MOZD.OutpFlowrateProduct;
NETWORK
TITLE = Calculate actual flowrate water
      L     -32767;
      L     #InpFlowrateWater;	//  kg/h
      >=I;
      AN    #Par.ParWago;	// Fault only with Siemens analog input
      S     #OutFaultAI;	//--> Overflow analog input
      L     0.000000e+00;
      JC    ai0;
      L     #InpFlowrateWater;	//  kg/h
      DTR;	// Integer to real
      L     #tmpMaxDigits;	// Units maximum         
      /R;
      L     #Par.ParFlowrateWater100Pc;
      DTR;	// Integer to real
      *R;
ai0:  T     #tmpFlowWater;
      RND;	// Real to Integer
      T     #OutFlowrateWater;
NETWORK
TITLE = Calculate Analog Output moisture
      L     0;
      AN    #StStarted;
      ON    #OutpRemote;
      JC    msJ1;
      L     #MYFA.InMoisture;	//[0.1%]
      DTR;	// Integer to real
      L     2.000000e+02;
      <=R;
      JC    msJ3;
      L     1.000000e+00;	// 100%          
      JU    msJ4;
msJ3: /R;
msJ4: L     #tmpMaxDigits;	// Units maximum         
      *R;
      RND;	// Real to Integer
msJ1: T     #MYFA.OutpMoisture;
NETWORK
TITLE = Calculate actual moisture
      L     -32767;
      L     #MYFA.InpMoisture;	//  
      >=I;
      AN    #Par.ParWago;	// Fault only with Siemens analog input
      S     #OutFaultAI;	//--> Overflow analog input
      L     0.000000e+00;
      JC    aim0;
      L     #MYFA.InpMoisture;	//  
      DTR;	// Integer to real
      L     #tmpMaxDigits;	// Units maximum         
      /R;
      L     2.000000e+02;
      *R;
aim0: RND;	// Real to Integer
      T     #MYFA.OutMoisture;
NETWORK
TITLE = BOTH: Calculate actual flowrate product
      L     -32767;
      L     #MYFA.InpFlowrateProduct;
      >=I;
      AN    #Par.ParWago;	// Fault only with Siemens analog input
      S     #OutFaultAI;	//--> Overflow analog input
      L     0.000000e+00;
      JC    aip0;
      L     #MYFA.InpFlowrateProduct;
      DTR;	// Integer to real
      L     #tmpMaxDigits;	// Units maximum         
      /R;
      L     #Par.ParFlowrateProduct100Pc;
      DTR;	// Integer to real
      *R;
aip0: RND;	// Real to Integer
      T     #MYFA.OutFlowrateProduct;
NETWORK
TITLE = BOTH: Calculate OutWtTotal
      AN    #CmdNewJob;
      JC    wtJ1;
      L     0;
      T     #OutTotalWater;
      L     0.000000e+00;
      T     #Par.OutCorrectionWeight;
      JU    clJ1;
wtJ1: AN    "GCS7_Gr_OutTick1s";	//Gr.OutTick1s
      JC    clJ1;
      L     #tmpFlowWater;
      L     3.600000e+03;	// [3600s]  
      /R;
      L     #Par.OutCorrectionWeight;
      +R;
      T     #Par.OutCorrectionWeight;
      RND-;
      L     #OutTotalWater;
      +D;
      T     #OutTotalWater;
      L     #Par.OutCorrectionWeight;
      L     #Par.OutCorrectionWeight;
      RND-;
      DTR;	// Integer to Real
      -R;
      T     #Par.OutCorrectionWeight;	//New rest 
NETWORK
TITLE = Global End
//---Clear all commands
clJ1: SET;
      R     #CmdOn;
      R     #CmdOff;
      R     #CmdNewJob;
      R     #CmdNext;
      R     #CmdFaultReset;
//--Output for group 
      A     #InDPFault;
      AN    #tmpLocalFault;
      S     "GCS7_Gr_InDPFault";
      A     #InHWStop;
      AN    #tmpLocalFault;
      S     "GCS7_Gr_InHWStop";
      A     #StFault;
      S     "GCS7_Gr_InFault";	// Gr.InFault
NETWORK
TITLE = State Code
//--Stopped, Substate ---
      AN    #StStopped;
      JC    STC2;
      L     41;	//Code: StStopped.HWStop
      A     #InHWStop;
      JC    STC;
      L     51;	//Code: StStopped.DPFault
      A     #InDPFault;
      JC    STC;
      L     1;	//Code: stopped
      A     #StStopped;
      JC    STC;
//===============
STC2: L     3;	// Code: started
      A     #StStarted;
      JC    STC;
      L     32;	// Code: fault
STC:  L     #StCode;	// Old state code
      TAK;
      T     #StCode;	// Save state code
      <>I;
      L     3;	// Load code for CBit methode
      CC    "SYS_CBitCtrl";
END_FUNCTION_BLOCK

FUNCTION_BLOCK "GCS7_E_Scale"	// FB 40
TITLE = Scale DIFF/DUMP
//  
//COPYRIGHT:    (C) 1996  BUHLER AG, CH-9240 UZWIL, SWITZERLAND
//
//PRODUCT:      GCS7
//
//TITLE:        Element Control Scale DIFF, DUMP, with OPTO22 or DP
//
//-------------------------------------------------------------------------
//
//IDENT:        AUTHOR:             DEPT:                       DATE:
//FB40.7.8      A. Egli             BASE                        29-Jan-2009
//              - DUMP Check InPreCutoffWeight and Status.TotalReached       
//FB40.7.7      Ph. Engler          GP92                        16-Jun-2008
//              - No failure with MEAG-Fault 17       
//              - Transition from StEmptying to StStarting when
//                InOutRestDischargeBin has been reset
//FB40.7.6      A. Egli             BASE                        09-Apr-2008
//              Disable Alarm 18 Battery Low
//FB40.7.5      A. Egli             CT3                         25-Mai-2007
//              - Overflow weight OutNotErasableWeight is 999'999'999 
//FB40.7.4      A.Egli              CT3                         20-Feb-2006
//              For CmdRefill test also tmpOn: Tested by P.Engler
//FB40.7.3      A.Egli              CT3                         01-Dec-2005
//              Parameter Upload Change DBD86-->DBD88
//FB40.7.2      A.Egli              CT3                         17-Mai-2005
//              Reset Flowrate only when OutComFault=1 
//FB40.7.1      A.Egli              CT3                         14-Mar-2005
//              Read Status.TotalReached only with data set 1
//FB40.7.0      A.Egli              CT3                         05-Jan-2005
//              Parameter Upload (uses DB10)
//FB40.6.6      Ph. Engler          MU664                       13-Sep-2004
//              -DIFF: Command.Restdischarge only in LCStep=1
//FB40.6.5      A.Egli              CT3                         23-Jul-2004
//              DUMP: Transition StDosing to StSopped also in LCStep=2
//FB40.6.4      A.Egli              CT3                         18-Mai-2004
//              DUMP: Transition to Started, when Level uncovered
//FB40.6.3      A.Egli              CT3                         24-Mar-2004
//              Replace T D [AR1,xxx] with T LD [AR1,xxx]
//FB40.6.2      A.Egli              CT3                         17-Nov-2003
//              - Alarm 90: Fault Remote Control
//              - MEAF: Ignor SumFault
//              - Local Mode: ComFault change to StStopped
//              - Manual mode: Set EnableEmptying
//FB40.6.1      A. Egli             CT3                         19-Mai-2003
//              Use Status.Operation as condtion for stopped
//FB40.6.0      A. Egli             CT3                         17-Jun-2002
//              New Release with one block
//              OPTO22 and Profibus   
//              LC Alarm 14 (DPFault) =Log Text number 12
//              InRecipeNr=Byte21
//FB40.5.1      P.Engler            CT3                         22-Mai-2002
//              Transition StStopped to StEmptying
//FB40.5.0      K.Tischer           CT3                         20-Sep-2001
//              Several modifications for MEAF
//FB40.4.3      K.Tischer           CT3                         02-Aug-2001
//              InSeqStopDUMP: S/R #OutStateTarget.EmptyingDUMP [4.3]
//FB40.4.2      A.Egli              CT3                         25-Jun-2001
//              par.OutLCAlarm.NoProduct replaced par.OutLCAlarm.NoProduct
//              Reset CmdRefill        
//FB40.4.1      P.Müller            MU664                       16-Mar-2001
//              Wait in StStarting until LCStep <> 1 removed
//FB40.4.0      S. Kalberer         CT3                         28-Nov-2000
//              Emptying event and signals adapted (MEAF V32B)
//FB40.3.0      A. Egli             CT3                         14-Jul-2000
//              New command MEAF
//FB40.2.6      A. Egli             CT3                         17-Mar-2000
//              Length for answer telegram
//FB40.2.4      S. Kalberer         CT3                         18-Feb-2000
//              CmdNewJob: Clear scale total in StDosing by OutStopPoint
//FB40.2.3      S. Kalberer         CT3                         11-Feb-2000
//              Relog fault, store OutState.InDischarged
//              CmdNewJob: immediate clear OutWtJobActual
//FB40.2C       S. Kalberer         CT3                         24-Sep-1999
//              Powerfailure dependency eliminated
//              ParManual behaviour corrected
//FB40.2B       S. Kalberer         CT3                         10-Mar-1999
//              MEAF compatible interface
//FB40.2A       A. Egli             CT3                         04-Mai-1998
//              StFault = StCode 32
//FB40.1A       A.Egli              AEE61                       28-Jul-1997
//              1st Release in S7
//
//-------------------------------------------------------------------------
//
//PURPOSE:      MANUAL : see [SCALExxMAN]
//
//RESTRICTIONS: S7
//              ACCU2: Pointer to dynamic datas of the element
//              ACCU1: Pointer to parameter datas of the element
//
//=======================================================
//Log Message: 
//------------------------------------------------------
//0     = Fault Cannceled
//1..79 = AlarmLC : Alarmnumber see manual of MEAF
//90    = Fault Remote Control
//91    = StStopped
//92    = StDosing
//93    = StEmptied
//94    = Timeout starting
//95    = WrongValue
//96    = Communication fault
//97    = 
//98    = 
//99    = Collected alarm
//
//=======================================================
//StCode:  State               
//------------------------------------------------------
//32   StFault                 
// 1   StStopped               
//41   StStopped.HWStop              StStopped + InHWStop 
//51   StStopped.DPFault             StStopped + DPFault
// 2   StStarting              
// 3   StDosing                
// 9   StEmptying              
//10   StEmptied               
//11   StRefill                
AUTHOR : EA
FAMILY : GCS7LL
NAME : SCALE
VERSION : 7.8
VAR
  StCode : INT ;	//Element state code
  InEnable : BOOL ;	//Enable to run scale
  InOutRestdischargeScale : BOOL ;	//Fully emptying scale (MEAF-DIFF)
  InDisableDischargeDUMP : BOOL ;	//stop discharge DUMP Scale
  InRestDosing : BOOL ;	//Restdosing (only MEAF)
  CmdNewValue : BOOL ;	//Send new taregt value to scale
  CmdNewJob : BOOL ;	//Clear actual weight or restart in state StEmptied
  CmdRefill : BOOL ;	//Refill of scale after maintenance (MEAF-DIFF)
  InOutRestdischargeBin : BOOL ;	//Fully emptying bin and scale (MEAF-DIFF + DUMP)
  CmdOff : BOOL ;	//Pulse to stop scale (manual mode)
  CmdOn : BOOL ;	//Pulse to start scale(manual mode)
  CmdNext : BOOL ;	//Start next element  (automatic mode)
  CmdFaultReset : BOOL ;	//Command to reset fault
  InLocal : BOOL ;	//1= Local mode (no fault by start with service switch)
  InManual : BOOL ;	//1= Manual/ 0= Automatic
  InReport : BOOL ;	//Report of all state transitions
  InSeqStopDUMP : BOOL ;	//Sequence stop scale by fully emptying scale (MEAF-DUMP)
  InHWStop : BOOL ;	//HW stop is detected, no fault
  InDPFault : BOOL ;	//DP-Fault is detected, no fault
  InSimulation : BOOL ;	//Simulation with DPSim
  OutComFault : BOOL ;	//Communication fault
  OutDepotEmpty : BOOL ;	//Alarm "DepotEmpty" is set (MEAF-DIFF)
  OutRefillDone : BOOL ;	//Refill is done (MEAF-DIFF)
  OutEmptied : BOOL ;	//Emptying is done
  OutpEnable : BOOL ;	//Output signale for scale
  StStopped : BOOL ;	//Element is stopped
  StStarting : BOOL ;	//Element is starting
  StDosing : BOOL ;	//Element is started, ready for dosing
  StEmptying : BOOL ;	//Emptying is active
  StFault : BOOL ;	//Element has a fault
  StEmptied : BOOL ;	//Element is emptied
  StRefill : BOOL ;	//Refill of the scale (MEAF-DIFF)
  spare57 : BOOL ;
  OutStopPoint : BOOL ;	//Target weight reached
  OutWeightCleared : BOOL ;	//Erasable weight is cleared
  OutWrongValue : BOOL ;	//Wrong nominal values, rejected by MEAF
  InFlowrate : DINT ;	//Is send to LC
  InJobWeight : DINT ;	//Is send to LC
  InRecipeNr : INT ;	//Is send to LC (DIFF only)
  InPreCutoffWeight : INT ;	//Pre cutoff weight
  OutFlowrate : DINT ;	//Is read from LC
  OutJobWeight : DINT ;	//Is calculated by element out of not erasable weight
  OutTotalWeight : DINT ;	//Is read from LC
  OutScaleWeight : DINT ;	//Is read from LC
  OutRecipeNr : INT ;	//Is read from LC (DIFF only)
  OutLCStep : INT ;	//Is read from LC
  OutAlarmNr : INT ;	//Is read from LC
  spare : DINT ;
  OutAlarmNrLog : INT ;	//Last textnumber send to log
  DUMP : STRUCT 	//DUMP only (is only sent, if InDumpWt >0)
   InDumpWeight : INT ;	//de: Schüttgrösse (only Profibus DP)
   InFlowrateLowLimit : INT ;	//de: Untere Leistungsgrenze
   InFlowrateHighLimit : INT ;	//de: Obere Leistungsgrenze
   spare : DINT ;
  END_STRUCT ;
  RecipeDiff : STRUCT 	//Recipe Diff Scale (Profibus only)
   InRecipeNr : INT ;	//Recipe to read or write (DIFF only)
   CmdSend : BOOL ;	//1= Send Dataset 136
   CmdRead : BOOL ;	//1= Read Dataset 136
   OutSendDone : BOOL ;	//Send is done
   OutReadDone : BOOL ;	//Read is done
   OutWrongValue : BOOL ;	//MEAF has recipe rejected
   InOutCutoffWeight : INT ;	//DIFF: Pre cutoff weight
   InOutDensity : INT ;	//DIFF: de: spezifisches Gewicht
   InOutFactor : INT ;	//DIFF: de: Verstaerkungsfaktor Dosiergeschwindigkeit
   InOutAutoCorrFactor : INT ;	//DIFF: de: Automatischer Korrektur Verstaerkungsfaktor
   spare : DINT ;
  END_STRUCT ;
  Par : STRUCT
   ParObjectNo : INT ;	//Is used for communication with PC, e.g. for message
   ParMsgType : INT ;	//Is used for message (translation of state)
   ParHornCode : INT ;	//Is used by horn module
   ParLogOff : BOOL ;	//Report is off
   ParManual : BOOL ;	//Manual mode without interlocking
   ParDUMP : BOOL ;	//1= MEAF:DUMP (MWEE)/ 0=MEAF:DIFF (MWEG,MWEY)
   ParOPTO22 : BOOL ;	//1= OPTO22 / 0= Profibus
   ParNoStep : BOOL ;	//OPTO22: Do not read command 'c' (MWEG1, MWEJ)
   ParMEAF : BOOL ;	//OPTO22: Use new MEAF commands, not compatible to old electronics
   ParFilter : STRUCT 	//Filter to alarm 1=Ignore alarm
    SumFault : BOOL ;	//All: de: Sammelalarm
    A05_24VToLow : BOOL ;	//All:
    A07ADRange : BOOL ;
    A08ADCalibration : BOOL ;
    A09ADFunction : BOOL ;
    A10ADSupply : BOOL ;
    A11AnalogInput : BOOL ;
    AxxCommunication : BOOL ;	//A12: Serial Interface ; A14=DPFault
    A13RemoteControl : BOOL ;
    A16Printer : BOOL ;
    A20NoStandStill : BOOL ;
    A21EmptyingTime : BOOL ;
    A22ScaleOpen : BOOL ;
    A23LLScaleHopper : BOOL ;
    A24WeightHopper : BOOL ;
    A25FrequenceConverter : BOOL ;
    A26Tolerance : BOOL ;
    A27Measurment : BOOL ;
    A28Feeddrive : BOOL ;
    A29FeedingTime : BOOL ;
    A30ZeroTara : BOOL ;
    A32InletSlideGate : BOOL ;
    A33AirPressure : BOOL ;
    A34NoProduct : BOOL ;
   END_STRUCT ;
   ParComDB : INT ;	//OPTO22: Communication DB
   ParLCIdx : INT ;	//OPTO22: Index of data record
   ParLCAddr : INT ;	//OPTO22: Address of LC
   ParIOByteNr : INT ;	//PROFIBUS: Address of first input and output byte Profibus DP
   ParMonTime : INT ;	//After this time the scale must be in the requested state (New)
   Spare90 : DINT ;
   Spare94 : DINT ;
   OutMonTime : INT ;
   OutScaleType : INT ;	//Is read from LC
   OutNotErasableWeight : DINT  := L#-1;	//Is read from LC
   HelpFlags : STRUCT 	//Aux. signal to retry fault message
    CmdNewValue : BOOL ;
    CmdNewJob : BOOL ;
    OutFaultResetDone : BOOL ;
    OutTestNewAlarm : BOOL ;
    CmdSend129 : BOOL ;	//Send of datablock 129 is requested
    OutFlagFaultResetDone : BOOL ;
    OutTargetSnd : BOOL ;
    OutStepRcv : BOOL ;
    OutAlarmTimeOut : BOOL ;
    EnableDosing : BOOL ;	//Help flag for immediate stop
    OutRelevantFault : BOOL ;
    OutNoAlarm : BOOL ;	//Alarmnumber 0 is read form LC
    OutComFaultRead : BOOL ;
    OutComFaultSend : BOOL ;
   END_STRUCT ;
   Command : STRUCT 	//Command for LC, is send to LC
    Start : BOOL ;	//de: Start
    ResetWtTotal : BOOL ;	//de: Total löschen
    RestDischarge : BOOL ;	//de: Restentleeren
    RestDosing_Refill : BOOL ;	//de: DUMP Restdosieren ; DIFF Refill
    EnableEmptying : BOOL ;	//de: Entleerfreigabe
    OverwriteLL : BOOL ;	//de: DIFF: Kein Alarm bei Leerstand
    spare06 : BOOL ;
    AcceptNewDataReady : BOOL ;	//de: Quittierung neue Werte Bereit
    spare10 : BYTE ;
    spare20 : BYTE ;
    CommandReady : BOOL ;	//de: Steuersignale gültig
    spare41 : BOOL ;
    spare42 : BOOL ;
    spare43 : BOOL ;
    spare44 : BOOL ;
    ResetAlarm : BOOL ;	//de: Alarm löschen
    NewSendData : BOOL ;	//de: Aenderung Sendedaten
    AcceptNewRcvData : BOOL ;	//de: Quittierung Aenderung Empfangsdatensatz
   END_STRUCT ;
   Status : STRUCT 	//MEAF DIFF
    Operation : BOOL ;	//de: Betrieb
    TotalReached : BOOL ;	//de: Total erreicht
    RestDischargeDone : BOOL ;	//de: Restentleeren ausgefüht
    PreCutoffWt_ReadyDosing : BOOL ;	//de: DUMP:Vorabschaltpunkt erreicht/DIFF:Dosierbereit
    TotalReady : BOOL ;	//de: Total bereit
    EnableFeeding_Empty : BOOL ;	//de: DUMP:Transportfreigabe/DIFF:Vordepot leer
    WeightPulse : BOOL ;	//de: Gewichtsimpuls
    NewDataReady : BOOL ;	//de: Neue Werte Bereit
    OutOfTolerance_LL : BOOL ;	//de: DUMP: Ausserhalb Leistungstoleranz/DIFF: Leerstand Waage
    _Dosingtime : BOOL ;	//de: DUMP: not used/DIFF: Dosierzeit ueberschritten
    _ZeroTolerance : BOOL ;	//de: DUMP: not used/DIFF: Niveau
    _RefillRequest : BOOL ;	//de: DUMP: not used/DIFF: Produktzufuehrung
    spare14 : BOOL ;
    spare15 : BOOL ;
    spare16 : BOOL ;
    spare17 : BOOL ;
    spare20 : BYTE ;
    Powerfailure : BOOL ;	//DIFF de: Power failure (only with old electronics)
    spare31 : BOOL ;
    spare32 : BOOL ;	//de: Stuerung Remote
    RemoteControlDP : BOOL ;	//de: Sollwertvorgabe Remote
    WrongValue : BOOL ;	//de: Falscher Sollwert
    SumFault : BOOL ;	//de: Sammelalarm
    AcceptNewSendData : BOOL ;	//de: Quittierung Aenderung Sendedaten
    NewRcvData : BOOL ;	//de: Aenderung Empfangsdaten
   END_STRUCT ;
   ComFlags : STRUCT 	//Flags for communication
    c_Done : BOOL ;	//step
    f_Done : BOOL ;	//Alarm, flowrate, actual weight (MEAF:DUMP)
    g_Done : BOOL ;	//Not erasible weight
    r_Done : BOOL ;	//Actual status
    t_Done : BOOL ;	//scale type
    w_Done : BOOL ;	//scale weight    (MEAF:DIFF)
    d_Done : BOOL ;	//Actual value 2  (MEAF:DIFF)
    h_Done : BOOL ;	//only MEAF
    U_Done : BOOL ;	//Lower  flow rate       (MEAF:DUMP)
    O_Done : BOOL ;	//Limit  upper flow rate (MEAF:DUMP)
    M_Done : BOOL ;	//Target weight
    Q_Done : BOOL ;	//Target flow rate
    S_Done : BOOL ;	//Target status 1
    TT_Done : BOOL ;	//Target status 2 (MEAF:DIFF)
    A_Done : BOOL ;	//Commands MEAF
    p_Done : BOOL ;	//not used
    PP_Done : BOOL ;	//not used
    CC_Done : BOOL ;	//C: DumpWt  (MEAF:DUMP)
   END_STRUCT ;
  END_STRUCT ;
END_VAR
VAR_TEMP
  tmpLOGvalue : WORD ;	//LOG value
  tmpCommand : INT ;
  tmpFBNO : INT ;	//Number of the actual FB
  tmpReport : BOOL ;	//Global LOG all
  tmpFault : BOOL ;
  tmpLocal : BOOL ;
  tmpClearCmdFlag : BOOL ;	//Clear pattern Commands
  tmpOn : BOOL ;
  tmpOff : BOOL ;
  tmpSeqStopDUMP : BOOL ;
  tmpWeight : DINT ;
  tmpLenDyn : DINT ;
  tmpAddrOutComFlags : DWORD ;	//Pointer to OutComFlags
  tmpComDB : INT ;
  tmpLocalFault : BOOL ;
  tmpAddrOffset : DINT ;
  tmpImmediateStop : BOOL ;
  tmpFilter : ARRAY  [0 .. 100 ] OF BOOL ;
  tmpAlarmDUMP : STRUCT 	//Is read from DUMP with command f
   Tolerance : BOOL ;	//Tolerance (not on collective alarm)
   SumFault : BOOL ;	//de: Sammelalarm ab V26A
   spare12 : BOOL ;	//n.w.
   ProbeScaleHopper : BOOL ;	//Probe scale hopper   -->alarm 23
   ScaleOpen : BOOL ;	//Scale open -->alarm 22
   StandStill : BOOL ;	//no standstill -->alarm 20
   EmptyingTime : BOOL ;	//emptying time -->alarm 21
   ADConverter : BOOL ;	//AD converter -->alarm 9
  END_STRUCT ;
  tmpAlarmDIFF : STRUCT 	//Is read from DIFF with command d
   DepotEmpty : BOOL ;	//Surge hopper empty (not on collect alarm) --> alarm 34
   ScaleEmpty : BOOL ;	//de: Leerstand Waage (no product)
   Discharger : BOOL ;	//DIFF a2 Frequency converter or feeding drive -->alarm 25
   Tolerance : BOOL ;	//DIFF a2 Tolerance --> alarm 26
   SumFault : BOOL ;	//de: Sammelalarm ab V26A
   TaraPos : BOOL ;	//DIFF a1 n.w.  -->alarm 30
   ADConverter : BOOL ;	//DIFF a1 AD converter--> alarm 9
   Reading : BOOL ;	//DIFF a1 Measuring fault --> alarm 27
  END_STRUCT ;
  tmpCommand_r : STRUCT 	//Is read from DUMP with command r
   Remote : BOOL ;	//MEAF DUMP: r1 Overiding operation
   DischargeDone : BOOL ;	//de: Restentleeren ausgefüht
   WtTotalReached : BOOL ;	//de: Total erreicht
  END_STRUCT ;
  tmpCommand_d : STRUCT 	//Is read from DIFF with command d
   log_1 : BOOL ;	//de: Always 1
   local : BOOL ;	//de: Local Operation
   DischargeDone : BOOL ;	//de: Restentleeren ausgefüht
   Cycle : BOOL ;	//de: Alters the state after every cycle
   Powerfailure : BOOL ;	//de: Power failure
   Operation : BOOL ;	//de: Betrieb (only with old electronic)
   WtTotalReached : BOOL ;	//de: Total erreicht
   ReadyDosing : BOOL ;	//de: Ready for Feeding
  END_STRUCT ;
  tmpCommand_S_DIFF : STRUCT 	//Command are sent to DIFF with command  S
   ResetPowerfailure : BOOL ;	//de:Stromausfallflg löschen
   EnableDosing : BOOL ;	//de: Dosierfreigabe
   ResetWtTotal : BOOL ;	//de: Total löschen
   Bit3 : BOOL ;	//not used
  END_STRUCT ;
  tmpCommand_T : STRUCT 	//Command are sent to DIFF with command  S and T
   Refill : BOOL ;	//fill up
   Emptying : BOOL ;	//discharge
   Bit2 : BOOL ;	//not used
   Bit3 : BOOL ;	//not used
  END_STRUCT ;
  tmpCommand_S_DUMP : STRUCT 	//Command are sent to DUMP with command  S
   RestDosing : BOOL ;	//de: Redsosieren ab V32B
   EnableDosing : BOOL ;	//de: Dosierfreigabe
   ResetWtTotal : BOOL ;	//de: Total löschen
   Emptying : BOOL ;	//de: Restentleeren
  END_STRUCT ;
  tmpCommand_A : STRUCT 	//Is send to MEAF with Command A
   ResetDischarge : BOOL ;	//DIFF:discharge       DUMP:Rest feeding
   StopDischarge_Restdosing : BOOL ;	//DIFF:Stop discharge  DUMP:Rest discharge
   Refill : BOOL ;	//DIFF:Fill up         DUMP:not used
   spare23 : BOOL ;	//
   Start : BOOL ;	//
   Stop : BOOL ;	//
   ResetWtTotal : BOOL ;	//de: Total löschen
   ResetAlarm : BOOL ;
   spare40 : BOOL ;	//
   spare41 : BOOL ;	//
   spare42 : BOOL ;	//
   Modify : BOOL ;	//DIFF/DUMP take over data
   spare30 : BOOL ;	//
   spare31 : BOOL ;	//
   spare32 : BOOL ;	//
   Modify2 : BOOL ;	//
  END_STRUCT ;
  tmpStatus_h_DUMP : STRUCT
   PreCutoffWt : BOOL ;	//de: Vorabschaltgewicht erreicht
   DischargeDone : BOOL ;	//de: Restentleeren ausgefüht
   spare22 : BOOL ;	//not used
   SumFault : BOOL ;	//de: Sammelalarm ab V26A
   Remote : BOOL ;	//de:
   NewDataReady : BOOL ;	//de: Neue Werte Bereit
   WtTotalReached : BOOL ;	//de: Total erreicht
   Tolerance : BOOL ;	//de: Ausserhalb Toleranz
  END_STRUCT ;
  tmpStatus_h_DIFF : STRUCT
   DischargeDone : BOOL ;	//de: Restentleeren ausgefüht
   BufferHopperEmpty : BOOL ;	//de: Vordepot leer
   ReadyDosing : BOOL ;	//de: Dosierbereit
   SumFault : BOOL ;	//de: Sammelalarm ab V26A
   Remote : BOOL ;	//de:
   NewDataReady : BOOL ;	//de: Neue Werte Bereit
   WtTotalReached : BOOL ;	//de: Total erreicht
   ScaleEmpty : BOOL ;	//de: Leerstand Waage (no product)
  END_STRUCT ;
  tmpAddr : WORD ;
  tmpReturn : INT ;
  Set136 : STRUCT
   Density : INT ;	//DIFF: de: spezifisches Gewicht
   Factor : INT ;	//DIFF: de: Verstaerkungsfaktor Dosiergeschwindigkeit
   CutoffWt : INT ;	//Pre cutoff weight
   spare14 : DINT ;
   spare18 : DINT ;
   spare22 : BYTE ;
   AutoCorrFactor : BYTE ;	//DIFF: de: Automatischer Korrektur Verstaerkungsfaktor
  END_STRUCT ;
  Set001 : STRUCT
   FlowrateAc : DINT ;	//de: Istleistung kg/h
   WtTotalAc : DINT ;	//de: Isttotalgewicht kg
   WtNotErasable : DINT ;	//de: nochtlöschbarese Totalgewicht
   spare12 : BYTE ;
   RecipeNr : BYTE ;
   Step : BYTE ;
   AlarmNr : BYTE ;
  END_STRUCT ;
  DPData : STRUCT
   StatusCommand : DWORD ;
   NrSndDataSet : BYTE ;	//de: Nummer Sendedatensatz
   IdxSndDataSet : BYTE ;	//de: Index Sendedatensatz
   NrRcvDataSet : BYTE ;	//de: Nummer Empfangsdatensatz
   IdxRcvDataSet : BYTE ;	//de: Index Empfangsdatensatz
   Data : ARRAY  [1 .. 4 ] OF DINT ;
  END_STRUCT ;
  tmpMEAF : BOOL ;
  tmpTotalReached : BOOL ;
  tmpDecPoint : INT ;
END_VAR
BEGIN
NETWORK
TITLE =  Start Global
      L     40;
      T     #tmpFBNO;
      L     126;
      T     #tmpLenDyn;	//--> Len dynamic data in byte
      TAR2;
      L     DW#16#FFFFFF;
      AD;
      T     #tmpAddrOffset;
      L     P##Par;
      +D;
      T     #tmpAddrOffset;
      L     P#48.0;
      +D;
      T     #tmpAddrOutComFlags;	// P##Par.ComFlags
      L     #Par.ParComDB;
      T     #tmpComDB;
      A     #Par.ParMEAF;
      ON    #Par.ParOPTO22;
      =     #tmpMEAF;
NETWORK
TITLE = Filter
      LAR1  P##tmpFilter;
      L     0;
      T     LD [AR1,P#0.0];	//tmpFilter[00..31]    [6.3]
      T     LD [AR1,P#0.0];	//tmpFilter[32..63]    [6.3]
      T     LD [AR1,P#0.0];	//tmpFilter[64..95]    [6.3]
      A     #Par.ParFilter.SumFault;
      O     #Par.ParMEAF;	//[6.2]
      =     #tmpFilter[0];
      A     #Par.ParFilter.A05_24VToLow;
      =     #tmpFilter[5];
      A     #Par.ParFilter.A07ADRange;
      =     #tmpFilter[7];
      A     #Par.ParFilter.A08ADCalibration;
      =     #tmpFilter[8];
      A     #Par.ParFilter.A09ADFunction;
      =     #tmpFilter[9];
      A     #Par.ParFilter.A10ADSupply;
      =     #tmpFilter[10];
      A     #Par.ParFilter.A11AnalogInput;
      =     #tmpFilter[11];
      A     #Par.ParFilter.AxxCommunication;
      =     #tmpFilter[12];
      =     #tmpFilter[14];
      A     #Par.ParFilter.A13RemoteControl;
      =     #tmpFilter[13];
      A     #Par.ParFilter.A16Printer;
      =     #tmpFilter[16];
      SET;
      =     #tmpFilter[17];	//[7.7]
      =     #tmpFilter[18];	//[7.6] Battery Low
      A     #Par.ParFilter.A20NoStandStill;
      =     #tmpFilter[20];
      A     #Par.ParFilter.A21EmptyingTime;
      =     #tmpFilter[21];
      A     #Par.ParFilter.A22ScaleOpen;
      =     #tmpFilter[22];
      A     #Par.ParFilter.A23LLScaleHopper;
      =     #tmpFilter[23];
      A     #Par.ParFilter.A24WeightHopper;
      =     #tmpFilter[24];
      A     #Par.ParFilter.A25FrequenceConverter;
      =     #tmpFilter[25];
      A     #Par.ParFilter.A26Tolerance;
      =     #tmpFilter[26];
      A     #Par.ParFilter.A27Measurment;
      =     #tmpFilter[27];
      A     #Par.ParFilter.A28Feeddrive;
      =     #tmpFilter[28];
      A     #Par.ParFilter.A29FeedingTime;
      =     #tmpFilter[29];
      A     #Par.ParFilter.A30ZeroTara;
      =     #tmpFilter[30];
      A     #Par.ParFilter.A32InletSlideGate;
      =     #tmpFilter[32];
      A     #Par.ParFilter.A33AirPressure;
      =     #tmpFilter[33];
      A     #Par.ParFilter.A34NoProduct;
      =     #tmpFilter[34];
      A     #InOutRestdischargeBin;	//[4.0]
      AN    #Par.ParDUMP;	//[4.0] DIFF scale only
      S     #tmpFilter[34];	//DepotEmpty
      S     #tmpFilter[24];	//NoProduct
      S     #tmpFilter[0];	//CollectedAlarm
NETWORK
TITLE = (OPTO22) Call back function
//*****This functio are called by FBxxx (COM) ******
//**********************************
//(OPTO22)
//**********************************
      AN    #Par.ParOPTO22;
      JC    O22A;
      OPN   DB [#tmpComDB];
      L     0;
      L     DBW 32;	//COM.Element.CODE;
      ==I;
      JC    PC;
      L     DBB 76;	//COM.Telegram.Command;
      T     #tmpCommand;
      L     1;
      L     DBW 32;	//COM.Element.CODE;
      ==I;
      JC    Send;
      L     2;
      ==I;
      JC    Rcv;
      L     4;	//NAK
      L     DBW 32;	//COM.Element.CODE;
      <>I;
      BEC;
      S     #OutComFault;
      BEU;
//===== Prepare data for send =================================
//Read telegram length
Send: L     #tmpCommand;
      L     'c';
      ==I;
      L     2;	//Lenght in byte
      JC    Sndx;
      L     #tmpCommand;
      L     'f';
      ==I;
      L     16;	//Lenght in byte
      JC    Sndx;
      L     #tmpCommand;
      L     'g';
      ==I;
      L     8;	//Lenght in byte
      JC    Sndx;
      L     #tmpCommand;
      L     'r';
      ==I;
      L     1;	//Lenght in byte
      JC    Sndx;
      L     #tmpCommand;
      L     't';
      ==I;
      L     2;	//Lenght in byte
      JC    Sndx;
      L     #tmpCommand;
      L     'w';
      ==I;
      L     6;	//Lenght in byte
      JC    Sndx;
      L     #tmpCommand;
      L     'd';
      ==I;
      L     18;	//Lenght in byte
      JC    Sndx;
      L     #tmpCommand;
      L     'h';
      ==I;
      L     36;	//Lenght in byte
      JC    Sndx;
      JU    SndA;
Sndx: T     DBW 86;	//COM.Telegram.LenAnswer
      JU    STOR;
//--------------------
//Send A [3.0]
//--------------------
SndA: L     #tmpCommand;
      L     'A';
      <>I;
      JC    SndM;
      LAR1  P##tmpCommand_A;
      L     0;
      T     LW [AR1,P#0.0];	//-->Reset tmpStateTarget
// command 1
      AN    #Par.Command.ResetWtTotal;	//[4.0]
      A     #Par.Command.Start;
      =     #tmpCommand_A.Start;
      A     #Par.Command.ResetWtTotal;	//[4.0]
      ON    #Par.Command.Start;
      =     #tmpCommand_A.Stop;
      A     #Par.Command.ResetWtTotal;	//[4.0]
      =     #tmpCommand_A.ResetWtTotal;	//[4.0]
      A     #Par.Command.ResetAlarm;
      =     #tmpCommand_A.ResetAlarm;
      R     #Par.Command.ResetAlarm;
      S     #Par.HelpFlags.OutFaultResetDone;
// command 2
      A     #Par.Command.RestDischarge;
      =     #tmpCommand_A.ResetDischarge;	//Restdischarge or Emptying                   //[5.0]
      A     #Par.Command.RestDosing_Refill;	//Rest Fedding after target weight is reached //[5.0]
      A     #Par.ParDUMP;	//                                                  //[5.0]
      O;	//                                                  //[5.0]
      AN    #Par.Command.RestDischarge;
      AN    #Par.ParDUMP;
      =     #tmpCommand_A.StopDischarge_Restdosing;
      A     #Par.Command.RestDosing_Refill;
      AN    #Par.ParDUMP;
      =     #tmpCommand_A.Refill;
// command 3
      SET;
      =     #tmpCommand_A.Modify;
// command 4
      =     #tmpCommand_A.Modify2;
//command 1..4
      L     0;	//Character offset
      T     DBW 40;	//COM.Element.AddrOffset
      LAR1  P##tmpCommand_A;
      L     LW [AR1,P#0.0];
      T     DBD 36;	//COM.Element.InOutValue
      L     34;	//Convert Hex to 4-ASCII
      T     DBW 0;	//COM.CODE
      CDB;	//ComDB->Instanz-DB
      UC    "GCS7_RS485Ctrl";	//Convert (CODE=DBW0)
      CDB;	//ElementDB->Instanz-DB
// RecipeNr   
      L     4;	//Character offset
      T     DBW 40;	//COM.Element.AddrOffset
      L     #InRecipeNr;
      T     DBD 36;	//COM.Element.InOutValue
      L     12;	//Convert DInt to 2-ASCII
      T     DBW 0;	//COM.CODE
      CDB;	//ComDB->Instanz-DB
      UC    "GCS7_RS485Ctrl";	//Convert (CODE=DBW0)
      CDB;	//ElementDB->Instanz-DB
// Flowrate    
      L     6;	//Character offset
      T     DBW 40;	//COM.Element.AddrOffset
      L     #InFlowrate;	//[4.0]
      T     DBD 36;	//COM.Element.InOutValue
      L     16;	//Convert DInt to 6-ASCII
      T     DBW 0;	//COM.CODE
      CDB;	//ComDB->Instanz-DB
      UC    "GCS7_RS485Ctrl";	//Convert (CODE=DBW0)
      CDB;	//ElementDB->Instanz-DB
// JobWeight    
      L     12;	//Character offset
      T     DBW 40;	//COM.Element.AddrOffset
      A     #InOutRestdischargeBin;
      AN    #Par.ParDUMP;
      L     0;
      JC    SA2;
      L     #InJobWeight;	//[4.0]
SA2:  T     DBD 36;	//COM.Element.InOutValue
      L     18;	//Convert DInt to 8-ASCII
      T     DBW 0;	//COM.CODE
      CDB;	//ComDB->Instanz-DB
      UC    "GCS7_RS485Ctrl";	//Convert (CODE=DBW0)
      CDB;	//ElementDB->Instanz-DB
      L     20;	//Lenght in byte
      T     DBW 78;	//COM.Telegram.Len
      JU    SndX;
//--------------------
//Send 'M'
//--------------------
SndM: L     #tmpCommand;
      L     'M';
      <>I;
      JC    SndO;
      L     #InJobWeight;	//[4.0]
      T     DBD 36;	//COM.Element.InOutValue
      L     18;	//Convert DInt to 6-ASCII
      T     DBW 0;	//COM.CODE
      CDB;	//ComDB->Instanz-DB
      UC    "GCS7_RS485Ctrl";	//Convert (CODE=DBW0)
      CDB;	//ElementDB->Instanz-DB
      L     8;	//Lenght in Byte
      JU    Snd1;
//--------------------
//Send 'O'
//--------------------
SndO: L     #tmpCommand;
      L     'O';
      <>I;
      JC    SndC;
      L     #DUMP.InFlowrateHighLimit;
      JU    Sd6;
//--------------------
//Send 'C'
//--------------------
SndC: L     #tmpCommand;
      L     'C';
      <>I;
      JC    SndU;
      L     #DUMP.InDumpWeight;
      T     DBD 36;	//COM.Element.InOutValue
      L     13;	//Convert DInt to 3-ASCII
      T     DBW 0;	//COM.CODE
      CDB;	//ComDB->Instanz-DB
      UC    "GCS7_RS485Ctrl";	//Convert (CODE=DBW0)
      CDB;	//ElementDB->Instanz-DB
      L     3;	//Lenght in Byte
      JU    Snd1;
//--------------------
//Send 'U'
//--------------------
SndU: L     #tmpCommand;
      L     'U';
      <>I;
      JC    SndQ;
      L     #DUMP.InFlowrateLowLimit;
      JU    Sd6;
//--------------------
//Send 'Q'
//--------------------
SndQ: L     #tmpCommand;
      L     'Q';
      <>I;
      JC    SndS;
      L     #InFlowrate;	//[4.0]
Sd6:  T     DBD 36;	//COM.Element.InOutValue
      L     16;	//Convert DInt to 6-ASCII
      T     DBW 0;	//COM.CODE
      CDB;	//ComDB->Instanz-DB
      UC    "GCS7_RS485Ctrl";	//Convert (CODE=DBW0)
      CDB;	//ElementDB->Instanz-DB
      L     6;	//Lenght in Byte
      JU    Snd1;
//--------------------
//Send 'S'
//--------------------
SndS: L     #tmpCommand;
      L     'S';
      <>I;
      JC    SndT;
      A     #Par.Command.ResetAlarm;
      R     #Par.Command.ResetAlarm;
      S     #Par.HelpFlags.OutFaultResetDone;
      A     #Par.ParDUMP;
      JC    SSDU;
      A     #OutpEnable;
      =     #Par.Command.Start;
      SET;
      =     #tmpCommand_S_DIFF.ResetPowerfailure;
      A     #OutpEnable;
      =     #tmpCommand_S_DIFF.EnableDosing;
      A     #Par.Command.ResetWtTotal;
      =     #tmpCommand_S_DIFF.ResetWtTotal;
      CLR;
      =     #tmpCommand_S_DIFF.Bit3;
      LAR1  P##tmpCommand_S_DIFF;
      L     LB [AR1,P#0.0];
      JU    sd1;
SSDU: NOP   0;
      A     #Par.Command.RestDosing_Refill;
      =     #tmpCommand_S_DUMP.RestDosing;
      A     #Par.Command.Start;
      =     #tmpCommand_S_DUMP.EnableDosing;
      A     #Par.Command.ResetWtTotal;
      =     #tmpCommand_S_DUMP.ResetWtTotal;
      A     #Par.Command.RestDischarge;
      =     #tmpCommand_S_DUMP.Emptying;
      LAR1  P##tmpCommand_S_DUMP;
      L     LB [AR1,P#0.0];
      JU    sd1;
//----Send 'T'
SndT: L     #tmpCommand;
      L     'T';
      <>I;
      JC    SndX;
      A     #Par.Command.RestDosing_Refill;
      =     #tmpCommand_T.Refill;
      A     #Par.Command.RestDischarge;
      =     #tmpCommand_T.Emptying;
      CLR;
      =     #tmpCommand_T.Bit2;
      =     #tmpCommand_T.Bit3;
      LAR1  P##tmpCommand_T;
      L     LB [AR1,P#0.0];
sd1:  T     DBD 36;	//COM.Element.InOutValue
      L     31;	//Convert Hex to 1ASCII
      T     DBW 0;	//COM.CODE
      CDB;	//ComDB->Instanz-DB
      UC    "GCS7_RS485Ctrl";	//Convert (CODE=DBW0)
      CDB;	//ElementDB->Instanz-DB
      A(;
      L     #OutLCStep;	//Step 1 = Init
      L     1;
      ==I;
      );
      A     #Par.Command.RestDischarge;	//[5.0]
      S     #Par.HelpFlags.OutTargetSnd;	//[5.0]
      L     1;	//Lenght in Byte
Snd1: T     DBW 78;	//COM.Telegram.Len; 
SndX: JU    STOR;
//======================================================================
//Answer Telegramm: Copy reveived data to element
//======================================================================
//--------------------
//Receive h [3.0]
//--------------------
Rcv:  R     #OutComFault;
      L     #tmpCommand;
      L     'h';
      <>I;
      JC    Rcvc;
      A     #Par.HelpFlags.OutFaultResetDone;	//[5.0]
      R     #Par.HelpFlags.OutFaultResetDone;	//[5.0]
      S     #Par.HelpFlags.OutTestNewAlarm;	//[5.0]
//State Actual                                                     //[5.0]
      SET;
      R     #Par.Status.Powerfailure;
      L     0;	//Character offset         //[5.0]
      T     DBW 40;	//ERH.Element.AddrOffset   //[5.0]
      L     42;	//Convert 2-ASCII to Hex   //[5.0]
      T     DBW 0;	//ERH.CODE                 //[5.0]
      CDB;	//ComDB->Instanz-DB        //[5.0]
      UC    "GCS7_RS485Ctrl";	//Convert (CODE=DBW0)      //[5.0]
      CDB;	//ElementDB->Instanz-DB    //[5.0]
      A     #Par.ParDUMP;	//                         //[6.0]
      JC    DUMP;	//                         //[6.0]
      L     DBD 36;	//ERH.Element.InOutValue   //[6.0]
      LAR1  P##tmpStatus_h_DIFF;	//[6.0]
      T     LB [AR1,P#0.0];	//-->#tmpStatus_h_DIFF       //[6.0]
      A     #tmpStatus_h_DIFF.DischargeDone;
      =     #Par.Status.RestDischargeDone;
      A     #tmpStatus_h_DIFF.BufferHopperEmpty;
      =     #Par.Status.EnableFeeding_Empty;
      A     #tmpStatus_h_DIFF.ReadyDosing;
      =     #Par.Status.PreCutoffWt_ReadyDosing;
      A     #tmpStatus_h_DIFF.SumFault;
      =     #Par.Status.SumFault;
      A     #tmpStatus_h_DIFF.Remote;
      =     #Par.Status.RemoteControlDP;
      A     #tmpStatus_h_DIFF.NewDataReady;
      =     #Par.Status.NewDataReady;
      A     #tmpStatus_h_DIFF.WtTotalReached;
      =     #Par.Status.TotalReached;
      A     #tmpStatus_h_DIFF.ScaleEmpty;
      =     #Par.Status.OutOfTolerance_LL;
      JU    NDUM;	//                         //[6.0]
DUMP: NOP   0;	//                         //[6.0]
      L     DBD 36;	//ERH.Element.InOutValue   //[6.0]
      LAR1  P##tmpStatus_h_DUMP;	//                         //[6.0]
      T     LB [AR1,P#0.0];	//-->#tmpStatus_h_DUMP       //[6.0]
      A     #tmpStatus_h_DUMP.PreCutoffWt;
      =     #Par.Status.PreCutoffWt_ReadyDosing;
      A     #tmpStatus_h_DUMP.DischargeDone;
      =     #Par.Status.RestDischargeDone;
      A     #tmpStatus_h_DUMP.SumFault;
      =     #Par.Status.SumFault;
      A     #tmpStatus_h_DUMP.Remote;
      =     #Par.Status.RemoteControlDP;
      A     #tmpStatus_h_DUMP.NewDataReady;
      =     #Par.Status.NewDataReady;
      A     #tmpStatus_h_DUMP.WtTotalReached;
      =     #Par.Status.TotalReached;
      A     #tmpStatus_h_DUMP.Tolerance;
      =     #Par.Status.OutOfTolerance_LL;
NDUM: NOP   0;	//                         //[6.0]
//StepNr
      L     2;	//Character offset
      T     DBW 40;	//COM.Element.AddrOffset
      L     22;	//Convert 2-ASCII to DInt
      T     DBW 0;	//COM.CODE
      CDB;	//ComDB->Instanz-DB
      UC    "GCS7_RS485Ctrl";	//Convert (CODE=DBW0)
      CDB;	//ElementDB->Instanz-DB
      L     DBD 36;	//COM.Element.InOutValue
      T     #OutLCStep;
//OutAlarmNr
      L     4;	//Character offset
      T     DBW 40;	//COM.Element.AddrOffset
      L     22;	//Convert 2-ASCII to DInt
      T     DBW 0;	//COM.CODE
      CDB;	//ComDB->Instanz-DB
      UC    "GCS7_RS485Ctrl";	//Convert (CODE=DBW0)
      CDB;	//ElementDB->Instanz-DB
      L     DBD 36;	//COM.Element.InOutValue
      T     #OutAlarmNr;
//Acutal flowrate
      L     6;	//Character offset
      T     DBW 40;	//COM.Element.AddrOffset
      L     26;	//Convert 6-ASCII to DInt
      T     DBW 0;	//COM.CODE
      CDB;	//ComDB->Instanz-DB
      UC    "GCS7_RS485Ctrl";	//Convert (CODE=DBW0)
      CDB;	//ElementDB->Instanz-DB
      L     DBD 36;	//COM.Element.InOutValue
      T     #OutFlowrate;	//[4.0]
//ScaleWeight
      L     12;	//Character offset
      T     DBW 40;	//COM.Element.AddrOffset
      L     26;	//Convert 6-ASCII to DInt
      T     DBW 0;	//ERH.CODE
      CDB;	//ComDB->Instanz-DB
      UC    "GCS7_RS485Ctrl";	//Convert (CODE=DBW0)
      CDB;	//ElementDB->Instanz-DB
      L     DBD 36;	//ERH.Element.InOutValue
      T     #OutScaleWeight;	//[4.0]
//- OutErasableWeight
      L     18;	//Character offset
      T     DBW 40;	//ERH.Element.AddrOffset
      L     28;	//Convert 8-ASCII to DInt
      T     DBW 0;	//ERH.CODE
      CDB;	//ComDB->Instanz-DB
      UC    "GCS7_RS485Ctrl";	//Convert (CODE=DBW0)
      CDB;	//ElementDB->Instanz-DB
      L     DBD 36;	//ERH.Element.InOutValue
      T     #OutTotalWeight;	//[4.0]
//Not erasable total
      L     26;	//Character offset
      T     DBW 40;	//COM.Element.AddrOffset
      L     28;	//Convert 8-ASCII to DInt
      T     DBW 0;	//COM.CODE
      CDB;	//ComDB->Instanz-DB
      UC    "GCS7_RS485Ctrl";	//Convert (CODE=DBW0)
      CDB;	//ElementDB->Instanz-DB
      L     DBD 36;	//COM.Element.InOutValue
      T     #tmpWeight;
      JU    RdJ1;
//--------------------
//Receive 'c'
//--------------------
Rcvc: L     #tmpCommand;
      L     'c';
      <>I;
      JC    Rcvd;
      L     22;	//Convert 2-ASCII to DInt
      T     DBW 0;	//ERH.CODE
      CDB;	//ComDB->Instanz-DB
      UC    "GCS7_RS485Ctrl";	//Convert (CODE=DBW0)
      CDB;	//ElementDB->Instanz-DB
      L     DBD 36;	//ERH.Element.InOutValue
      T     #OutLCStep;
      A     #Par.HelpFlags.OutTargetSnd;	//[5.0]
      S     #Par.HelpFlags.OutStepRcv;	//[5.0]
      JU    STOR;
//--------------------
//Receive 'd'
//--------------------
Rcvd: L     #tmpCommand;
      L     'd';
      <>I;
      JC    Rcvf;
      A     #Par.HelpFlags.OutFaultResetDone;
      R     #Par.HelpFlags.OutFaultResetDone;
      S     #Par.HelpFlags.OutTestNewAlarm;
//- OutState
      L     42;	//Convert 2-ASCII to Hex
      T     DBW 0;	//ERH.CODE
      CDB;	//ComDB->Instanz-DB
      UC    "GCS7_RS485Ctrl";	//Convert (CODE=DBW0)
      CDB;	//ElementDB->Instanz-DB
      L     DBD 36;	//ERH.Element.InOutValue
      LAR1  P##tmpCommand_d;
      T     LB [AR1,P#0.0];	//-->#tmpStatusDIFF;
      AN    #tmpCommand_d.local;
      =     #Par.Status.RemoteControlDP;
      A     #tmpCommand_d.DischargeDone;
      =     #Par.Status.RestDischargeDone;
      A     #tmpCommand_d.Powerfailure;
      =     #Par.Status.Powerfailure;
      A     #tmpCommand_d.Operation;
      =     #Par.Status.Operation;
      A     #tmpCommand_d.WtTotalReached;
      =     #Par.Status.TotalReached;
      A     #tmpCommand_d.ReadyDosing;
      =     #Par.Status.PreCutoffWt_ReadyDosing;
//- OutLCAlarm
      L     2;	//Character offset
      T     DBW 40;	//ERH.Element.AddrOffset
      L     42;	//Convert 2-ASCII to Hex
      T     DBW 0;	//ERH.CODE
      CDB;	//ComDB->Instanz-DB
      UC    "GCS7_RS485Ctrl";	//Convert (CODE=DBW0)
      CDB;	//ElementDB->Instanz-DB
      L     DBD 36;	//ERH.Element.InOutValue
      LAR1  P##tmpAlarmDIFF;
      T     LB [AR1,P#0.0];	//-->#tmpAlarmDIFF;
//- OutFlowRate
      L     4;	//Character offset
      T     DBW 40;	//ERH.Element.AddrOffset
      L     26;	//Convert 6-ASCII to DInt
      T     DBW 0;	//ERH.CODE
      CDB;	//ComDB->Instanz-DB
      UC    "GCS7_RS485Ctrl";	//Convert (CODE=DBW0)
      CDB;	//ElementDB->Instanz-DB
      L     DBD 36;	//ERH.Element.InOutValue
      T     #OutFlowrate;	//[4.0]
//- OutErasableWeight
      L     10;	//Character offset
      T     DBW 40;	//ERH.Element.AddrOffset
      L     28;	//Convert 8-ASCII to DInt
      T     DBW 0;	//ERH.CODE
      CDB;	//ComDB->Instanz-DB
      UC    "GCS7_RS485Ctrl";	//Convert (CODE=DBW0)
      CDB;	//ElementDB->Instanz-DB
      L     DBD 36;	//ERH.Element.InOutValue
      T     #OutTotalWeight;	//[4.0]
//[6.0--->] Convert DIFF-Alarm to AlarmNr 
      A     #tmpAlarmDIFF.DepotEmpty;
      =     #Par.Status.EnableFeeding_Empty;
      A     #tmpAlarmDIFF.ScaleEmpty;
      =     #Par.Status.OutOfTolerance_LL;
      A     #tmpAlarmDIFF.SumFault;
      =     #Par.Status.SumFault;
      L     24;
      A     #tmpAlarmDIFF.ScaleEmpty;
      JC    ALN2;
      L     25;
      A     #tmpAlarmDIFF.Discharger;
      JC    ALN2;
      L     26;
      A     #tmpAlarmDIFF.Tolerance;
      JC    ALN2;
      L     30;
      A     #tmpAlarmDIFF.TaraPos;
      JC    ALN2;
      L     9;
      A     #tmpAlarmDIFF.ADConverter;
      JC    ALN2;
      L     27;
      A     #tmpAlarmDIFF.Reading;
      JC    ALN2;
      L     34;
      A     #tmpAlarmDIFF.DepotEmpty;
      JC    ALN2;
      L     0;
ALN2: T     #OutAlarmNr;
      JU    STOR;
//-------------------
//Receive 'f'
//-------------------
Rcvf: L     #tmpCommand;
      L     'f';
      <>I;
      JC    Rcvg;
      A     #Par.HelpFlags.OutFaultResetDone;
      R     #Par.HelpFlags.OutFaultResetDone;
      S     #Par.HelpFlags.OutTestNewAlarm;
//- OutLCAlarm
      L     42;	//Convert 2-ASCII to Hex
      T     DBW 0;	//ERH.CODE
      CDB;	//ComDB->Instanz-DB
      UC    "GCS7_RS485Ctrl";	//Convert (CODE=DBW0)
      CDB;	//ElementDB->Instanz-DB
      L     DBD 36;	//ERH.Element.InOutValue
      LAR1  P##tmpAlarmDUMP;
      T     LB [AR1,P#0.0];	//-->#tmpAlarmDUMP
//- OutFlowRate
      L     2;	//Character offset
      T     DBW 40;	//ERH.Element.AddrOffset
      L     26;	//Convert 6-ASCII to DInt
      T     DBW 0;	//ERH.CODE
      CDB;	//ComDB->Instanz-DB
      UC    "GCS7_RS485Ctrl";	//Convert (CODE=DBW0)
      CDB;	//ElementDB->Instanz-DB
      L     DBD 36;	//ERH.Element.InOutValue
      T     #OutFlowrate;	//[4.0]
//- OutErasableWeight
      L     8;	//Character offset
      T     DBW 40;	//ERH.Element.AddrOffset
      L     28;	//Convert 8-ASCII to DInt
      T     DBW 0;	//ERH.CODE
      CDB;	//ComDB->Instanz-DB
      UC    "GCS7_RS485Ctrl";	//Convert (CODE=DBW0)
      CDB;	//ElementDB->Instanz-DB
      L     DBD 36;	//ERH.Element.InOutValue
      T     #OutTotalWeight;	//[4.0]
//[6.0--->] Convert DUMP-Alarm to AlarmNr 
      A     #tmpAlarmDUMP.SumFault;
      =     #Par.Status.SumFault;
      A     #tmpAlarmDUMP.Tolerance;
      =     #Par.Status.OutOfTolerance_LL;
      L     23;
      A     #tmpAlarmDUMP.ProbeScaleHopper;
      JC    ALNR;
      L     22;
      A     #tmpAlarmDUMP.ScaleOpen;
      JC    ALNR;
      L     20;
      A     #tmpAlarmDUMP.StandStill;
      JC    ALNR;
      L     21;
      A     #tmpAlarmDUMP.EmptyingTime;
      JC    ALNR;
      L     9;
      A     #tmpAlarmDUMP.ADConverter;
      JC    ALNR;
      L     0;
ALNR: T     #OutAlarmNr;
//[<--6.0] 
      JU    STOR;
//--------------------
//Receive 'g'
//--------------------
Rcvg: L     #tmpCommand;
      L     'g';
      <>I;
      JC    Rcvr;
//- OutErasableWeight
      L     28;	//Convert 8-ASCII to DInt
      T     DBW 0;	//ERH.CODE
      CDB;	//ComDB->Instanz-DB
      UC    "GCS7_RS485Ctrl";	//Convert (CODE=DBW0)
      CDB;	//ElementDB->Instanz-DB
      L     DBD 36;	//ERH.Element.InOutValue
      T     #tmpWeight;
//---  Init first, if old value < 0  ---
RdJ1: L     #Par.OutNotErasableWeight;	//[4.0]
      L     0;
      <D;
      JC    rgZ2;
//---  Calculate Weight ---
      L     #tmpWeight;
      L     #Par.OutNotErasableWeight;	//[4.0]
      -D;
      JM    rgZ1;
      JU    rgPo;
rgZ1: L     L#100000000;
      +D;
rgPo: L     10000;	// Maximum change by relaod software
      >D;
      JC    rgZ2;
      TAK;
      L     #OutJobWeight;	//[4.0]
      +D;
      T     #OutJobWeight;	//[4.0]--> Total weight
rgZ2: L     #tmpWeight;
      T     #Par.OutNotErasableWeight;	//[4.0]
      JU    STOR;
//--------------------
//Receive 'r'
//--------------------
Rcvr: L     #tmpCommand;
      L     'r';
      <>I;
      JC    Rcvt;
//- OutState
      L     41;	//Convert 1-ASCII to Hex
      T     DBW 0;	//ERH.CODE
      CDB;	//ComDB->Instanz-DB
      UC    "GCS7_RS485Ctrl";	//Convert (CODE=DBW0)
      CDB;	//ElementDB->Instanz-DB
      L     DBD 36;	//ERH.Element.InOutValue
      LAR1  P##tmpCommand_r;
      T     LB [AR1,P#0.0];	//-->#tmpCommand_r;
      A     #tmpCommand_r.Remote;
      =     #Par.Status.RemoteControlDP;
      A     #tmpCommand_r.DischargeDone;
      =     #Par.Status.RestDischargeDone;
      A     #tmpCommand_r.WtTotalReached;
      =     #Par.Status.TotalReached;
      JU    STOR;
//--------------------
//Receive 't': Type
//--------------------
Rcvt: L     #tmpCommand;
      L     't';
      <>I;
      JC    Rcvw;
      L     22;	//Convert 2-ASCII to DInt
      T     DBW 0;	//ERH.CODE
      CDB;	//ComDB->Instanz-DB
      UC    "GCS7_RS485Ctrl";	//Convert (CODE=DBW0)
      CDB;	//ElementDB->Instanz-DB
      L     DBD 36;	//ERH.Element.InOutValue
      T     #Par.OutScaleType;
      JU    STOR;
//--------------------
//Receive 'w': Scale Weight
//--------------------
Rcvw: L     #tmpCommand;
      L     'w';
      <>I;
      JC    RcvS;
      L     26;	//Convert 6-ASCII to DInt
      T     DBW 0;	//ERH.CODE
      CDB;	//ComDB->Instanz-DB
      UC    "GCS7_RS485Ctrl";	//Convert (CODE=DBW0)
      CDB;	//ElementDB->Instanz-DB
      L     DBD 36;	//ERH.Element.InOutValue
      T     #OutScaleWeight;	//[4.0]
      JU    STOR;
//--------------------
//Accept 'S','A'
//--------------------
RcvS: L     #tmpCommand;
      L     'S';
      <>I;
      A(;
      L     #tmpCommand;
      L     'A';
      <>I;
      );
      JC    STOR;
      AN    #Par.Command.ResetWtTotal;	//[4.0] 
      JC    STOR;
      L     #OutTotalWeight;	//[4.0]
      L     0;
      ==I;
      ON    #Par.ParMEAF;
      R     #Par.Command.ResetWtTotal;	//[4.0] 
      S     #OutWeightCleared;
      R     #Par.HelpFlags.CmdNewJob;
STOR: BEU;
O22A: NOP   0;
NETWORK
TITLE = PC Control
//=== Test Object number =====================
PC:   L     "SYS_DirectCtrlDB".PC.ObjectNo;	//PCControl.ObjectNo
      L     #Par.ParObjectNo;	//Input ObjectNo
      <>I;
      JC    Ctrl;
//=== Test OType      ========================
      L     1040;	//Input object type
      L     "SYS_DirectCtrlDB".PC.ObjectType;	//PCControl.ObjectType
      <>I;
      JC    Ctrl;
//=== Test Handshake =========================
      A     "SYS_DirectCtrlDB".PC.Hsk.FExamine;	//Handshake.FExamine
      JC    pExa;
      A     "SYS_DirectCtrlDB".PC.Hsk.FDefineCmd;	//Handshake.FDefineCmd
      JC    pCmd;
      A     "SYS_DirectCtrlDB".PC.Hsk.FDefinePara;	//Handshake.FDefinePara
      JC    pPar;
pIni: L     2;	//FcInit
      UC    "SYS_DirectCtrl";
      JU    Ctrl;
// Write parameter 
pPar: LAR1  P#DBX 58.0;
      L     P##Par;
      L     DW#16#FFFFF;
      AD;
      +AR1;
      L     DBD [AR1,P#20.0];
      T     #Par.ParMonTime;
//Write new commands from PC to Interface of group 
pCmd: A     "SYS_DirectCtrlDB".PC.Cmd1[2];	//Cmd1[2]  =CmdRestDosingOn
      S     #InRestDosing;
      A     "SYS_DirectCtrlDB".PC.Cmd2[2];	//Cmd1[2]  =CmdRestDosingOff
      R     #InRestDosing;
      A     "SYS_DirectCtrlDB".PC.Cmd1[4];	//Cmd1[4]  =CmdNewValue
      S     #CmdNewValue;
      A     "SYS_DirectCtrlDB".PC.Cmd1[5];	//Cmd1[5]  =CmdNewJob
      S     #CmdNewJob;
      A     "SYS_DirectCtrlDB".PC.Cmd1[6];	//Cmd1[6]  =CmdRefill  
      S     #CmdRefill;
      A     "SYS_DirectCtrlDB".PC.Cmd1[7];	//Cmd1[7]  =CmdEmptying
      S     #InOutRestdischargeBin;	//                         [5.0]
      A     "SYS_DirectCtrlDB".PC.Cmd1[8];	//Cmd1[8]  =CmdOff
      S     #CmdOff;
      A     "SYS_DirectCtrlDB".PC.Cmd1[9];	//Cmd1[9]  =CmdOn
      S     #CmdOn;
      A     "SYS_DirectCtrlDB".PC.Cmd1[10];	//Cmd1[10]=CmdNext
      S     #CmdNext;
      A     "SYS_DirectCtrlDB".PC.Cmd1[11];	//Cmd1[11]=CmdFaultReset
      S     #CmdFaultReset;
      A     "SYS_DirectCtrlDB".PC.Cmd1[13];	//Cmd1[13]=CmdManualOn
      S     #InManual;
      A     "SYS_DirectCtrlDB".PC.Cmd2[13];	//Cmd2[13]=CmdManualOff
      R     #InManual;
      A     "SYS_DirectCtrlDB".PC.Cmd1[14];	//Cmd1[14]=CmdReportOn
      S     #InReport;
      A     "SYS_DirectCtrlDB".PC.Cmd2[14];	//Cmd2[14]=CmdReportOff
      R     #InReport;
//Define Value
      AN    "SYS_DirectCtrlDB".PC.Hsk.FDefineValue;	// PC.Hsk.FDefineValue
      ON    #InManual;
      JC    pIni;
      LAR1  P#DBX 58.0;
      L     DBD [AR1,P#8.0];
      T     #InFlowrate;
      L     DBD [AR1,P#12.0];
      T     #InJobWeight;
      L     DBW [AR1,P#16.0];
      T     #InRecipeNr;
      L     DBW [AR1,P#18.0];
      T     #InPreCutoffWeight;
      L     DBW [AR1,P#48.0];
      T     #DUMP.InDumpWeight;
      L     DBW [AR1,P#52.0];
      T     #DUMP.InFlowrateLowLimit;
      L     DBW [AR1,P#54.0];
      T     #DUMP.InFlowrateHighLimit;
      JU    pIni;
pExa: TAR2;	//Address Dynamic datas
      T     "SYS_DirectCtrlDB".GC.InDynAddr;	//-->PCControl.GC.InDynAddr
      L     #tmpLenDyn;	//Length Dynamic datas
      T     "SYS_DirectCtrlDB".GC.InDynLen;	//-->PCControl.GC.InDynLen
      L     0;
      T     "SYS_DirectCtrlDB".GC.InParaAddr;	//-->PCControl.GC.InParaAddr
      T     "SYS_DirectCtrlDB".GC.InParaLen;	//-->PCControl.GC.InParaLen
      L     1;	//Code FcExamine
      UC    "SYS_DirectCtrl";
      L     10;	//Revision
      T     "SYS_DirectCtrlDB".GC.Revision;
Ctrl: NOP   0;
NETWORK
TITLE = [7.0] LCParameter
      L     #Par.ParObjectNo;
      L     "SYS_DirectCtrlLCDB".PC.ObjectNo;
      <>I;
      ON    #Par.ParOPTO22;
      JC    LCP0;
      T     "SYS_DirectCtrlLCDB".GC.InObjectNo;
      L     #Par.ParComDB;
      T     "SYS_DirectCtrlLCDB".GC.InDBNr;
      L     #Par.ParLCAddr;
      T     "SYS_DirectCtrlLCDB".GC.InLCAddr;
LCP0: NOP   0;
NETWORK
TITLE = (OPTO22) Read LC data
//**********************************
//(OPTO22)
//**********************************
      AN    #Par.ParOPTO22;
      JC    O22B;
      OPN   DB [#tmpComDB];
      L     #Par.ParLCIdx;
      T     DBW 34;	//COM.Element.Index; 
      L     1;	//Read LC data
      T     DBW 0;	//COM.CODE;
      CDB;
      UC    "GCS7_RS485Ctrl";
      CDB;
      L     #tmpFBNO;
      T     DBW 52;	//COM.LC0.FBNO;   
      L     DINO;
      T     DBW 54;	//COM.LC0.DINO;
      TAR2  DBD 56;	//COM.LC0.AddrDyn;        
      L     0;
      T     DBD 60;	//COM.LC0.AddrPara;       
      L     #Par.ParLCAddr;
      T     DBD 64;	//COM.Telegram.LCAddr;
O22B: NOP   0;
NETWORK
TITLE = (Profibus) Read data
//**********************************
//(Profibus)
//**********************************
      A     #Par.ParOPTO22;
      JC    DP_A;
      L     #Par.ParIOByteNr;
      T     #tmpAddr;
      A     #InSimulation;
      JC    rSim;
      CALL  "SIEMENS_DPRD_DAT" (
           LADDR                    := #tmpAddr,
           RET_VAL                  := #tmpReturn,
           RECORD                   := #DPData);
      L     #tmpReturn;
      L     0;
      <>I;
      =     #Par.HelpFlags.OutComFaultRead;
      JC    rcv0;
      JU    rDP;
//read from Simulation
rSim: R     #Par.HelpFlags.OutComFaultRead;
      A     "GCS7_Gr_SimDPtoImage";
      L     P#I 0.0;
      JC    rDB1;
      OPN   "TEST_IOSimuliInput";
      L     P#DBX 0.0;
rDB1: L     #Par.ParIOByteNr;
      SLD   3;
      +D;
      LAR1;
      L     D [AR1,P#0.0];
      T     #DPData.StatusCommand;
      L     B [AR1,P#4.0];
      T     #DPData.NrSndDataSet;
      L     B [AR1,P#5.0];
      T     #DPData.IdxSndDataSet;
      L     B [AR1,P#6.0];
      T     #DPData.NrRcvDataSet;
      L     B [AR1,P#7.0];
      T     #DPData.IdxRcvDataSet;
      L     D [AR1,P#8.0];
      T     #DPData.Data[1];
      L     D [AR1,P#12.0];
      T     #DPData.Data[2];
      L     D [AR1,P#16.0];
      T     #DPData.Data[3];
      L     D [AR1,P#20.0];
      T     #DPData.Data[4];
//==Copy Status===============
rDP:  L     #DPData.NrRcvDataSet;
      L     0;
      ==I;
      JC    R001;
      A     #Par.Status.TotalReached;	//[7.1]
      =     #tmpTotalReached;	//[7.1]
      CALL  "SIEMENS_BLKMOV" (
           SRCBLK                   := #DPData.StatusCommand,
           RET_VAL                  := #tmpReturn,
           DSTBLK                   := #Par.Status);
      A     #tmpTotalReached;	//[7.1]
      =     #Par.Status.TotalReached;	//[7.1]
      AN    #Par.Status.NewRcvData;
      A     #InSimulation;
      JC    rcv0;
//===============================
//Answer Dataset 001
      L     #DPData.NrRcvDataSet;
      L     1;
      <>I;
      JC    r11;	//[7.0]
      CALL  "SIEMENS_BLKMOV" (
           SRCBLK                   := #DPData.StatusCommand,
           RET_VAL                  := #tmpReturn,
           DSTBLK                   := #Par.Status);	//[7.1]
      CALL  "SIEMENS_BLKMOV" (
           SRCBLK                   := #DPData.Data,
           RET_VAL                  := #tmpReturn,
           DSTBLK                   := #Set001);
      L     #Set001.FlowrateAc;
      T     #OutFlowrate;
      L     #Set001.WtTotalAc;
